(* Logix 5000 project; controller reports 1756-L63 rev 20.11; software revision 20.04; part 25 of 52 *)

        [1708].log_data[0].total := 300.0, [1708].log_data[0].time := 300.0, [1708].log_data[0].minminute := 40, [1708].log_data[0].maxminute := 40, [1708].log_data[0].valid := 1, [1708].log_data[1].valid := 1, [1708].log_data[2].valid := 1, [1708].log_data[3].valid := 1, [1708].log_data[4].valid := 1, [1708].log_data[5].valid := 1, [1708].log_data[6].valid := 1, [1708].log_data[7].valid := 1, [1708].log_data[8].valid := 1, [1708].log_data[9].valid := 1, [1708].log_data[10].valid := 1, [1708].log_data[11].valid := 1, [1708].log_data[12].valid := 1, [1708].log_data[13].valid := 1, [1708].log_data[14].valid := 1, [1708].log_data[15].valid := 1, [1708].log_data[16].valid := 1, [1708].log_data[17].valid := 1, [1708].log_data[18].valid := 1, [1708].log_data[19].valid := 1, [1708].time.Year := 2023, [1708].time.Month := 1, [1708].time.Day := 15, [1708].time.Hour := 14, [1708].time.Minute := 44, [1708].time.Second := 59, [1709].log_data[0].min := 1.0, [1709].log_data[0].max := 1.0, [1709].log_data[0].total := 300.0, [1709].log_data[0].time := 300.0, [1709].log_data[0].minminute := 45, [1709].log_data[0].maxminute := 45, [1709].log_data[0].valid := 1, [1709].log_data[1].valid := 1, [1709].log_data[2].valid := 1, [1709].log_data[3].valid := 1, [1709].log_data[4].valid := 1, [1709].log_data[5].valid := 1, [1709].log_data[6].valid := 1, [1709].log_data[7].valid := 1, [1709].log_data[8].valid := 1, [1709].log_data[9].valid := 1, [1709].log_data[10].valid := 1, [1709].log_data[11].valid := 1, [1709].log_data[12].valid := 1, [1709].log_data[13].valid := 1, [1709].log_data[14].valid := 1, [1709].log_data[15].valid := 1, [1709].log_data[16].valid := 1, [1709].log_data[17].valid := 1, [1709].log_data[18].valid := 1, [1709].log_data[19].valid := 1, [1709].time.Year := 2023, [1709].time.Month := 1, [1709].time.Day := 15, [1709].time.Hour := 14,
        [1709].time.Minute := 49, [1709].time.Second := 59, [1710].log_data[0].min := 1.0, [1710].log_data[0].max := 1.0, [1710].log_data[0].total := 300.0, [1710].log_data[0].time := 300.0, [1710].log_data[0].minminute := 50, [1710].log_data[0].maxminute := 50, [1710].log_data[0].valid := 1, [1710].log_data[1].valid := 1, [1710].log_data[2].valid := 1, [1710].log_data[3].valid := 1, [1710].log_data[4].valid := 1, [1710].log_data[5].valid := 1, [1710].log_data[6].valid := 1, [1710].log_data[7].valid := 1, [1710].log_data[8].valid := 1, [1710].log_data[9].valid := 1, [1710].log_data[10].valid := 1, [1710].log_data[11].valid := 1, [1710].log_data[12].valid := 1, [1710].log_data[13].valid := 1, [1710].log_data[14].valid := 1, [1710].log_data[15].valid := 1, [1710].log_data[16].valid := 1, [1710].log_data[17].valid := 1, [1710].log_data[18].valid := 1, [1710].log_data[19].valid := 1, [1710].time.Year := 2023, [1710].time.Month := 1, [1710].time.Day := 15, [1710].time.Hour := 14, [1710].time.Minute := 54, [1710].time.Second := 59, [1711].log_data[0].min := 1.0, [1711].log_data[0].max := 1.0, [1711].log_data[0].total := 300.0, [1711].log_data[0].time := 300.0, [1711].log_data[0].minminute := 55, [1711].log_data[0].maxminute := 55, [1711].log_data[0].valid := 1, [1711].log_data[1].valid := 1, [1711].log_data[2].valid := 1, [1711].log_data[3].valid := 1, [1711].log_data[4].valid := 1, [1711].log_data[5].valid := 1, [1711].log_data[6].valid := 1, [1711].log_data[7].valid := 1, [1711].log_data[8].valid := 1, [1711].log_data[9].valid := 1, [1711].log_data[10].valid := 1, [1711].log_data[11].valid := 1, [1711].log_data[12].valid := 1, [1711].log_data[13].valid := 1, [1711].log_data[14].valid := 1, [1711].log_data[15].valid := 1, [1711].log_data[16].valid := 1, [1711].log_data[17].valid := 1, [1711].log_data[18].valid := 1, [1711].log_data[19].valid := 1,
        [1711].time.Year := 2023, [1711].time.Month := 1, [1711].time.Day := 15, [1711].time.Hour := 14, [1711].time.Minute := 59, [1711].time.Second := 59, [1712].log_data[0].min := 1.0, [1712].log_data[0].max := 1.0, [1712].log_data[0].total := 300.0, [1712].log_data[0].time := 300.0, [1712].log_data[0].valid := 1, [1712].log_data[1].valid := 1, [1712].log_data[2].valid := 1, [1712].log_data[3].valid := 1, [1712].log_data[4].valid := 1, [1712].log_data[5].valid := 1, [1712].log_data[6].valid := 1, [1712].log_data[7].valid := 1, [1712].log_data[8].valid := 1, [1712].log_data[9].valid := 1, [1712].log_data[10].valid := 1, [1712].log_data[11].valid := 1, [1712].log_data[12].valid := 1, [1712].log_data[13].valid := 1, [1712].log_data[14].valid := 1, [1712].log_data[15].valid := 1, [1712].log_data[16].valid := 1, [1712].log_data[17].valid := 1, [1712].log_data[18].valid := 1, [1712].log_data[19].valid := 1, [1712].time.Year := 2023, [1712].time.Month := 1, [1712].time.Day := 15, [1712].time.Hour := 15, [1712].time.Minute := 4, [1712].time.Second := 59, [1713].log_data[0].min := 1.0, [1713].log_data[0].max := 1.0, [1713].log_data[0].total := 300.0, [1713].log_data[0].time := 300.0, [1713].log_data[0].minminute := 5, [1713].log_data[0].maxminute := 5, [1713].log_data[0].valid := 1, [1713].log_data[1].valid := 1, [1713].log_data[2].valid := 1, [1713].log_data[3].valid := 1, [1713].log_data[4].valid := 1, [1713].log_data[5].valid := 1, [1713].log_data[6].valid := 1, [1713].log_data[7].valid := 1, [1713].log_data[8].valid := 1, [1713].log_data[9].valid := 1, [1713].log_data[10].valid := 1, [1713].log_data[11].valid := 1, [1713].log_data[12].valid := 1, [1713].log_data[13].valid := 1, [1713].log_data[14].valid := 1, [1713].log_data[15].valid := 1, [1713].log_data[16].valid := 1, [1713].log_data[17].valid := 1,
        [1713].log_data[18].valid := 1, [1713].log_data[19].valid := 1, [1713].time.Year := 2023, [1713].time.Month := 1, [1713].time.Day := 15, [1713].time.Hour := 15, [1713].time.Minute := 9, [1713].time.Second := 59, [1714].log_data[0].min := 1.0, [1714].log_data[0].max := 1.0, [1714].log_data[0].total := 300.0, [1714].log_data[0].time := 300.0, [1714].log_data[0].minminute := 10, [1714].log_data[0].maxminute := 10, [1714].log_data[0].valid := 1, [1714].log_data[1].valid := 1, [1714].log_data[2].valid := 1, [1714].log_data[3].valid := 1, [1714].log_data[4].valid := 1, [1714].log_data[5].valid := 1, [1714].log_data[6].valid := 1, [1714].log_data[7].valid := 1, [1714].log_data[8].valid := 1, [1714].log_data[9].valid := 1, [1714].log_data[10].valid := 1, [1714].log_data[11].valid := 1, [1714].log_data[12].valid := 1, [1714].log_data[13].valid := 1, [1714].log_data[14].valid := 1, [1714].log_data[15].valid := 1, [1714].log_data[16].valid := 1, [1714].log_data[17].valid := 1, [1714].log_data[18].valid := 1, [1714].log_data[19].valid := 1, [1714].time.Year := 2023, [1714].time.Month := 1, [1714].time.Day := 15, [1714].time.Hour := 15, [1714].time.Minute := 14, [1714].time.Second := 59, [1715].log_data[0].min := 1.0, [1715].log_data[0].max := 1.0, [1715].log_data[0].total := 300.0, [1715].log_data[0].time := 300.0, [1715].log_data[0].minminute := 15, [1715].log_data[0].maxminute := 15, [1715].log_data[0].valid := 1, [1715].log_data[1].valid := 1, [1715].log_data[2].valid := 1, [1715].log_data[3].valid := 1, [1715].log_data[4].valid := 1, [1715].log_data[5].valid := 1, [1715].log_data[6].valid := 1, [1715].log_data[7].valid := 1, [1715].log_data[8].valid := 1, [1715].log_data[9].valid := 1, [1715].log_data[10].valid := 1, [1715].log_data[11].valid := 1, [1715].log_data[12].valid := 1, [1715].log_data[13].valid := 1,
        [1715].log_data[14].valid := 1, [1715].log_data[15].valid := 1, [1715].log_data[16].valid := 1, [1715].log_data[17].valid := 1, [1715].log_data[18].valid := 1, [1715].log_data[19].valid := 1, [1715].time.Year := 2023, [1715].time.Month := 1, [1715].time.Day := 15, [1715].time.Hour := 15, [1715].time.Minute := 19, [1715].time.Second := 59, [1716].log_data[0].min := 1.0, [1716].log_data[0].max := 1.0, [1716].log_data[0].total := 300.0, [1716].log_data[0].time := 300.0, [1716].log_data[0].minminute := 20, [1716].log_data[0].maxminute := 20, [1716].log_data[0].valid := 1, [1716].log_data[1].valid := 1, [1716].log_data[2].valid := 1, [1716].log_data[3].valid := 1, [1716].log_data[4].valid := 1, [1716].log_data[5].valid := 1, [1716].log_data[6].valid := 1, [1716].log_data[7].valid := 1, [1716].log_data[8].valid := 1, [1716].log_data[9].valid := 1, [1716].log_data[10].valid := 1, [1716].log_data[11].valid := 1, [1716].log_data[12].valid := 1, [1716].log_data[13].valid := 1, [1716].log_data[14].valid := 1, [1716].log_data[15].valid := 1, [1716].log_data[16].valid := 1, [1716].log_data[17].valid := 1, [1716].log_data[18].valid := 1, [1716].log_data[19].valid := 1, [1716].time.Year := 2023, [1716].time.Month := 1, [1716].time.Day := 15, [1716].time.Hour := 15, [1716].time.Minute := 24, [1716].time.Second := 59, [1717].log_data[0].min := 1.0, [1717].log_data[0].max := 1.0, [1717].log_data[0].total := 300.0, [1717].log_data[0].time := 300.0, [1717].log_data[0].minminute := 25, [1717].log_data[0].maxminute := 25, [1717].log_data[0].valid := 1, [1717].log_data[1].valid := 1, [1717].log_data[2].valid := 1, [1717].log_data[3].valid := 1, [1717].log_data[4].valid := 1, [1717].log_data[5].valid := 1, [1717].log_data[6].valid := 1, [1717].log_data[7].valid := 1, [1717].log_data[8].valid := 1, [1717].log_data[9].valid := 1,
        [1717].log_data[10].valid := 1, [1717].log_data[11].valid := 1, [1717].log_data[12].valid := 1, [1717].log_data[13].valid := 1, [1717].log_data[14].valid := 1, [1717].log_data[15].valid := 1, [1717].log_data[16].valid := 1, [1717].log_data[17].valid := 1, [1717].log_data[18].valid := 1, [1717].log_data[19].valid := 1, [1717].time.Year := 2023, [1717].time.Month := 1, [1717].time.Day := 15, [1717].time.Hour := 15, [1717].time.Minute := 29, [1717].time.Second := 59, [1718].log_data[0].min := 1.0, [1718].log_data[0].max := 1.0, [1718].log_data[0].total := 300.0, [1718].log_data[0].time := 300.0, [1718].log_data[0].minminute := 30, [1718].log_data[0].maxminute := 30, [1718].log_data[0].valid := 1, [1718].log_data[1].valid := 1, [1718].log_data[2].valid := 1, [1718].log_data[3].valid := 1, [1718].log_data[4].valid := 1, [1718].log_data[5].valid := 1, [1718].log_data[6].valid := 1, [1718].log_data[7].valid := 1, [1718].log_data[8].valid := 1, [1718].log_data[9].valid := 1, [1718].log_data[10].valid := 1, [1718].log_data[11].valid := 1, [1718].log_data[12].valid := 1, [1718].log_data[13].valid := 1, [1718].log_data[14].valid := 1, [1718].log_data[15].valid := 1, [1718].log_data[16].valid := 1, [1718].log_data[17].valid := 1, [1718].log_data[18].valid := 1, [1718].log_data[19].valid := 1, [1718].time.Year := 2023, [1718].time.Month := 1, [1718].time.Day := 15, [1718].time.Hour := 15, [1718].time.Minute := 34, [1718].time.Second := 59, [1719].log_data[0].min := 1.0, [1719].log_data[0].max := 1.0, [1719].log_data[0].total := 300.0, [1719].log_data[0].time := 300.0, [1719].log_data[0].minminute := 35, [1719].log_data[0].maxminute := 35, [1719].log_data[0].valid := 1, [1719].log_data[1].valid := 1, [1719].log_data[2].valid := 1, [1719].log_data[3].valid := 1, [1719].log_data[4].valid := 1, [1719].log_data[5].valid := 1,
        [1719].log_data[6].valid := 1, [1719].log_data[7].valid := 1, [1719].log_data[8].valid := 1, [1719].log_data[9].valid := 1, [1719].log_data[10].valid := 1, [1719].log_data[11].valid := 1, [1719].log_data[12].valid := 1, [1719].log_data[13].valid := 1, [1719].log_data[14].valid := 1, [1719].log_data[15].valid := 1, [1719].log_data[16].valid := 1, [1719].log_data[17].valid := 1, [1719].log_data[18].valid := 1, [1719].log_data[19].valid := 1, [1719].time.Year := 2023, [1719].time.Month := 1, [1719].time.Day := 15, [1719].time.Hour := 15, [1719].time.Minute := 39, [1719].time.Second := 59, [1720].log_data[0].min := 1.0, [1720].log_data[0].max := 1.0, [1720].log_data[0].total := 300.0, [1720].log_data[0].time := 300.0, [1720].log_data[0].minminute := 40, [1720].log_data[0].maxminute := 40, [1720].log_data[0].valid := 1, [1720].log_data[1].valid := 1, [1720].log_data[2].valid := 1, [1720].log_data[3].valid := 1, [1720].log_data[4].valid := 1, [1720].log_data[5].valid := 1, [1720].log_data[6].valid := 1, [1720].log_data[7].valid := 1, [1720].log_data[8].valid := 1, [1720].log_data[9].valid := 1, [1720].log_data[10].valid := 1, [1720].log_data[11].valid := 1, [1720].log_data[12].valid := 1, [1720].log_data[13].valid := 1, [1720].log_data[14].valid := 1, [1720].log_data[15].valid := 1, [1720].log_data[16].valid := 1, [1720].log_data[17].valid := 1, [1720].log_data[18].valid := 1, [1720].log_data[19].valid := 1, [1720].time.Year := 2023, [1720].time.Month := 1, [1720].time.Day := 15, [1720].time.Hour := 15, [1720].time.Minute := 44, [1720].time.Second := 59, [1721].log_data[0].min := 1.0, [1721].log_data[0].max := 1.0, [1721].log_data[0].total := 300.0, [1721].log_data[0].time := 300.0, [1721].log_data[0].minminute := 45, [1721].log_data[0].maxminute := 45, [1721].log_data[0].valid := 1, [1721].log_data[1].valid := 1,
        [1721].log_data[2].valid := 1, [1721].log_data[3].valid := 1, [1721].log_data[4].valid := 1, [1721].log_data[5].valid := 1, [1721].log_data[6].valid := 1, [1721].log_data[7].valid := 1, [1721].log_data[8].valid := 1, [1721].log_data[9].valid := 1, [1721].log_data[10].valid := 1, [1721].log_data[11].valid := 1, [1721].log_data[12].valid := 1, [1721].log_data[13].valid := 1, [1721].log_data[14].valid := 1, [1721].log_data[15].valid := 1, [1721].log_data[16].valid := 1, [1721].log_data[17].valid := 1, [1721].log_data[18].valid := 1, [1721].log_data[19].valid := 1, [1721].time.Year := 2023, [1721].time.Month := 1, [1721].time.Day := 15, [1721].time.Hour := 15, [1721].time.Minute := 49, [1721].time.Second := 59, [1722].log_data[0].min := 1.0, [1722].log_data[0].max := 1.0, [1722].log_data[0].total := 300.0, [1722].log_data[0].time := 300.0, [1722].log_data[0].minminute := 50, [1722].log_data[0].maxminute := 50, [1722].log_data[0].valid := 1, [1722].log_data[1].valid := 1, [1722].log_data[2].valid := 1, [1722].log_data[3].valid := 1, [1722].log_data[4].valid := 1, [1722].log_data[5].valid := 1, [1722].log_data[6].valid := 1, [1722].log_data[7].valid := 1, [1722].log_data[8].valid := 1, [1722].log_data[9].valid := 1, [1722].log_data[10].valid := 1, [1722].log_data[11].valid := 1, [1722].log_data[12].valid := 1, [1722].log_data[13].valid := 1, [1722].log_data[14].valid := 1, [1722].log_data[15].valid := 1, [1722].log_data[16].valid := 1, [1722].log_data[17].valid := 1, [1722].log_data[18].valid := 1, [1722].log_data[19].valid := 1, [1722].time.Year := 2023, [1722].time.Month := 1, [1722].time.Day := 15, [1722].time.Hour := 15, [1722].time.Minute := 54, [1722].time.Second := 59, [1723].log_data[0].min := 1.0, [1723].log_data[0].max := 1.0, [1723].log_data[0].total := 300.0, [1723].log_data[0].time := 300.0,
        [1723].log_data[0].minminute := 55, [1723].log_data[0].maxminute := 55, [1723].log_data[0].valid := 1, [1723].log_data[1].valid := 1, [1723].log_data[2].valid := 1, [1723].log_data[3].valid := 1, [1723].log_data[4].valid := 1, [1723].log_data[5].valid := 1, [1723].log_data[6].valid := 1, [1723].log_data[7].valid := 1, [1723].log_data[8].valid := 1, [1723].log_data[9].valid := 1, [1723].log_data[10].valid := 1, [1723].log_data[11].valid := 1, [1723].log_data[12].valid := 1, [1723].log_data[13].valid := 1, [1723].log_data[14].valid := 1, [1723].log_data[15].valid := 1, [1723].log_data[16].valid := 1, [1723].log_data[17].valid := 1, [1723].log_data[18].valid := 1, [1723].log_data[19].valid := 1, [1723].time.Year := 2023, [1723].time.Month := 1, [1723].time.Day := 15, [1723].time.Hour := 15, [1723].time.Minute := 59, [1723].time.Second := 59, [1724].log_data[0].min := 1.0, [1724].log_data[0].max := 1.0, [1724].log_data[0].total := 300.0, [1724].log_data[0].time := 300.0, [1724].log_data[0].valid := 1, [1724].log_data[1].valid := 1, [1724].log_data[2].valid := 1, [1724].log_data[3].valid := 1, [1724].log_data[4].valid := 1, [1724].log_data[5].valid := 1, [1724].log_data[6].valid := 1, [1724].log_data[7].valid := 1, [1724].log_data[8].valid := 1, [1724].log_data[9].valid := 1, [1724].log_data[10].valid := 1, [1724].log_data[11].valid := 1, [1724].log_data[12].valid := 1, [1724].log_data[13].valid := 1, [1724].log_data[14].valid := 1, [1724].log_data[15].valid := 1, [1724].log_data[16].valid := 1, [1724].log_data[17].valid := 1, [1724].log_data[18].valid := 1, [1724].log_data[19].valid := 1, [1724].time.Year := 2023, [1724].time.Month := 1, [1724].time.Day := 15, [1724].time.Hour := 16, [1724].time.Minute := 4, [1724].time.Second := 59, [1725].log_data[0].min := 1.0, [1725].log_data[0].max := 1.0,
        [1725].log_data[0].total := 300.0, [1725].log_data[0].time := 300.0, [1725].log_data[0].minminute := 5, [1725].log_data[0].maxminute := 5, [1725].log_data[0].valid := 1, [1725].log_data[1].valid := 1, [1725].log_data[2].valid := 1, [1725].log_data[3].valid := 1, [1725].log_data[4].valid := 1, [1725].log_data[5].valid := 1, [1725].log_data[6].valid := 1, [1725].log_data[7].valid := 1, [1725].log_data[8].valid := 1, [1725].log_data[9].valid := 1, [1725].log_data[10].valid := 1, [1725].log_data[11].valid := 1, [1725].log_data[12].valid := 1, [1725].log_data[13].valid := 1, [1725].log_data[14].valid := 1, [1725].log_data[15].valid := 1, [1725].log_data[16].valid := 1, [1725].log_data[17].valid := 1, [1725].log_data[18].valid := 1, [1725].log_data[19].valid := 1, [1725].time.Year := 2023, [1725].time.Month := 1, [1725].time.Day := 15, [1725].time.Hour := 16, [1725].time.Minute := 9, [1725].time.Second := 59, [1726].log_data[0].min := 1.0, [1726].log_data[0].max := 1.0, [1726].log_data[0].total := 300.0, [1726].log_data[0].time := 300.0, [1726].log_data[0].minminute := 10, [1726].log_data[0].maxminute := 10, [1726].log_data[0].valid := 1, [1726].log_data[1].valid := 1, [1726].log_data[2].valid := 1, [1726].log_data[3].valid := 1, [1726].log_data[4].valid := 1, [1726].log_data[5].valid := 1, [1726].log_data[6].valid := 1, [1726].log_data[7].valid := 1, [1726].log_data[8].valid := 1, [1726].log_data[9].valid := 1, [1726].log_data[10].valid := 1, [1726].log_data[11].valid := 1, [1726].log_data[12].valid := 1, [1726].log_data[13].valid := 1, [1726].log_data[14].valid := 1, [1726].log_data[15].valid := 1, [1726].log_data[16].valid := 1, [1726].log_data[17].valid := 1, [1726].log_data[18].valid := 1, [1726].log_data[19].valid := 1, [1726].time.Year := 2023, [1726].time.Month := 1, [1726].time.Day := 15, [1726].time.Hour := 16,
        [1726].time.Minute := 14, [1726].time.Second := 59, [1727].log_data[0].min := 1.0, [1727].log_data[0].max := 1.0, [1727].log_data[0].total := 300.0, [1727].log_data[0].time := 300.0, [1727].log_data[0].minminute := 15, [1727].log_data[0].maxminute := 15, [1727].log_data[0].valid := 1, [1727].log_data[1].valid := 1, [1727].log_data[2].valid := 1, [1727].log_data[3].valid := 1, [1727].log_data[4].valid := 1, [1727].log_data[5].valid := 1, [1727].log_data[6].valid := 1, [1727].log_data[7].valid := 1, [1727].log_data[8].valid := 1, [1727].log_data[9].valid := 1, [1727].log_data[10].valid := 1, [1727].log_data[11].valid := 1, [1727].log_data[12].valid := 1, [1727].log_data[13].valid := 1, [1727].log_data[14].valid := 1, [1727].log_data[15].valid := 1, [1727].log_data[16].valid := 1, [1727].log_data[17].valid := 1, [1727].log_data[18].valid := 1, [1727].log_data[19].valid := 1, [1727].time.Year := 2023, [1727].time.Month := 1, [1727].time.Day := 15, [1727].time.Hour := 16, [1727].time.Minute := 19, [1727].time.Second := 59, [1728].log_data[0].min := 1.0, [1728].log_data[0].max := 1.0, [1728].log_data[0].total := 300.0, [1728].log_data[0].time := 300.0, [1728].log_data[0].minminute := 20, [1728].log_data[0].maxminute := 20, [1728].log_data[0].valid := 1, [1728].log_data[1].valid := 1, [1728].log_data[2].valid := 1, [1728].log_data[3].valid := 1, [1728].log_data[4].valid := 1, [1728].log_data[5].valid := 1, [1728].log_data[6].valid := 1, [1728].log_data[7].valid := 1, [1728].log_data[8].valid := 1, [1728].log_data[9].valid := 1, [1728].log_data[10].valid := 1, [1728].log_data[11].valid := 1, [1728].log_data[12].valid := 1, [1728].log_data[13].valid := 1, [1728].log_data[14].valid := 1, [1728].log_data[15].valid := 1, [1728].log_data[16].valid := 1, [1728].log_data[17].valid := 1, [1728].log_data[18].valid := 1, [1728].log_data[19].valid := 1,
        [1728].time.Year := 2023, [1728].time.Month := 1, [1728].time.Day := 15, [1728].time.Hour := 16, [1728].time.Minute := 24, [1728].time.Second := 59, [1729].log_data[0].min := 1.0, [1729].log_data[0].max := 1.0, [1729].log_data[0].total := 300.0, [1729].log_data[0].time := 300.0, [1729].log_data[0].minminute := 25, [1729].log_data[0].maxminute := 25, [1729].log_data[0].valid := 1, [1729].log_data[1].valid := 1, [1729].log_data[2].valid := 1, [1729].log_data[3].valid := 1, [1729].log_data[4].valid := 1, [1729].log_data[5].valid := 1, [1729].log_data[6].valid := 1, [1729].log_data[7].valid := 1, [1729].log_data[8].valid := 1, [1729].log_data[9].valid := 1, [1729].log_data[10].valid := 1, [1729].log_data[11].valid := 1, [1729].log_data[12].valid := 1, [1729].log_data[13].valid := 1, [1729].log_data[14].valid := 1, [1729].log_data[15].valid := 1, [1729].log_data[16].valid := 1, [1729].log_data[17].valid := 1, [1729].log_data[18].valid := 1, [1729].log_data[19].valid := 1, [1729].time.Year := 2023, [1729].time.Month := 1, [1729].time.Day := 15, [1729].time.Hour := 16, [1729].time.Minute := 29, [1729].time.Second := 59, [1730].log_data[0].min := 1.0, [1730].log_data[0].max := 1.0, [1730].log_data[0].total := 300.0, [1730].log_data[0].time := 300.0, [1730].log_data[0].minminute := 30, [1730].log_data[0].maxminute := 30, [1730].log_data[0].valid := 1, [1730].log_data[1].valid := 1, [1730].log_data[2].valid := 1, [1730].log_data[3].valid := 1, [1730].log_data[4].valid := 1, [1730].log_data[5].valid := 1, [1730].log_data[6].valid := 1, [1730].log_data[7].valid := 1, [1730].log_data[8].valid := 1, [1730].log_data[9].valid := 1, [1730].log_data[10].valid := 1, [1730].log_data[11].valid := 1, [1730].log_data[12].valid := 1, [1730].log_data[13].valid := 1, [1730].log_data[14].valid := 1, [1730].log_data[15].valid := 1,
        [1730].log_data[16].valid := 1, [1730].log_data[17].valid := 1, [1730].log_data[18].valid := 1, [1730].log_data[19].valid := 1, [1730].time.Year := 2023, [1730].time.Month := 1, [1730].time.Day := 15, [1730].time.Hour := 16, [1730].time.Minute := 34, [1730].time.Second := 59, [1731].log_data[0].min := 1.0, [1731].log_data[0].max := 1.0, [1731].log_data[0].total := 300.0, [1731].log_data[0].time := 300.0, [1731].log_data[0].minminute := 35, [1731].log_data[0].maxminute := 35, [1731].log_data[0].valid := 1, [1731].log_data[1].valid := 1, [1731].log_data[2].valid := 1, [1731].log_data[3].valid := 1, [1731].log_data[4].valid := 1, [1731].log_data[5].valid := 1, [1731].log_data[6].valid := 1, [1731].log_data[7].valid := 1, [1731].log_data[8].valid := 1, [1731].log_data[9].valid := 1, [1731].log_data[10].valid := 1, [1731].log_data[11].valid := 1, [1731].log_data[12].valid := 1, [1731].log_data[13].valid := 1, [1731].log_data[14].valid := 1, [1731].log_data[15].valid := 1, [1731].log_data[16].valid := 1, [1731].log_data[17].valid := 1, [1731].log_data[18].valid := 1, [1731].log_data[19].valid := 1, [1731].time.Year := 2023, [1731].time.Month := 1, [1731].time.Day := 15, [1731].time.Hour := 16, [1731].time.Minute := 39, [1731].time.Second := 59, [1732].log_data[0].min := 1.0, [1732].log_data[0].max := 1.0, [1732].log_data[0].total := 300.0, [1732].log_data[0].time := 300.0, [1732].log_data[0].minminute := 40, [1732].log_data[0].maxminute := 40, [1732].log_data[0].valid := 1, [1732].log_data[1].valid := 1, [1732].log_data[2].valid := 1, [1732].log_data[3].valid := 1, [1732].log_data[4].valid := 1, [1732].log_data[5].valid := 1, [1732].log_data[6].valid := 1, [1732].log_data[7].valid := 1, [1732].log_data[8].valid := 1, [1732].log_data[9].valid := 1, [1732].log_data[10].valid := 1, [1732].log_data[11].valid := 1,
        [1732].log_data[12].valid := 1, [1732].log_data[13].valid := 1, [1732].log_data[14].valid := 1, [1732].log_data[15].valid := 1, [1732].log_data[16].valid := 1, [1732].log_data[17].valid := 1, [1732].log_data[18].valid := 1, [1732].log_data[19].valid := 1, [1732].time.Year := 2023, [1732].time.Month := 1, [1732].time.Day := 15, [1732].time.Hour := 16, [1732].time.Minute := 44, [1732].time.Second := 59, [1733].log_data[0].min := 1.0, [1733].log_data[0].max := 1.0, [1733].log_data[0].total := 300.0, [1733].log_data[0].time := 300.0, [1733].log_data[0].minminute := 45, [1733].log_data[0].maxminute := 45, [1733].log_data[0].valid := 1, [1733].log_data[1].valid := 1, [1733].log_data[2].valid := 1, [1733].log_data[3].valid := 1, [1733].log_data[4].valid := 1, [1733].log_data[5].valid := 1, [1733].log_data[6].valid := 1, [1733].log_data[7].valid := 1, [1733].log_data[8].valid := 1, [1733].log_data[9].valid := 1, [1733].log_data[10].valid := 1, [1733].log_data[11].valid := 1, [1733].log_data[12].valid := 1, [1733].log_data[13].valid := 1, [1733].log_data[14].valid := 1, [1733].log_data[15].valid := 1, [1733].log_data[16].valid := 1, [1733].log_data[17].valid := 1, [1733].log_data[18].valid := 1, [1733].log_data[19].valid := 1, [1733].time.Year := 2023, [1733].time.Month := 1, [1733].time.Day := 15, [1733].time.Hour := 16, [1733].time.Minute := 49, [1733].time.Second := 59, [1734].log_data[0].min := 1.0, [1734].log_data[0].max := 1.0, [1734].log_data[0].total := 300.0, [1734].log_data[0].time := 300.0, [1734].log_data[0].minminute := 50, [1734].log_data[0].maxminute := 50, [1734].log_data[0].valid := 1, [1734].log_data[1].valid := 1, [1734].log_data[2].valid := 1, [1734].log_data[3].valid := 1, [1734].log_data[4].valid := 1, [1734].log_data[5].valid := 1, [1734].log_data[6].valid := 1, [1734].log_data[7].valid := 1,
        [1734].log_data[8].valid := 1, [1734].log_data[9].valid := 1, [1734].log_data[10].valid := 1, [1734].log_data[11].valid := 1, [1734].log_data[12].valid := 1, [1734].log_data[13].valid := 1, [1734].log_data[14].valid := 1, [1734].log_data[15].valid := 1, [1734].log_data[16].valid := 1, [1734].log_data[17].valid := 1, [1734].log_data[18].valid := 1, [1734].log_data[19].valid := 1, [1734].time.Year := 2023, [1734].time.Month := 1, [1734].time.Day := 15, [1734].time.Hour := 16, [1734].time.Minute := 54, [1734].time.Second := 59, [1735].log_data[0].min := 1.0, [1735].log_data[0].max := 1.0, [1735].log_data[0].total := 300.0, [1735].log_data[0].time := 300.0, [1735].log_data[0].minminute := 55, [1735].log_data[0].maxminute := 55, [1735].log_data[0].valid := 1, [1735].log_data[1].valid := 1, [1735].log_data[2].valid := 1, [1735].log_data[3].valid := 1, [1735].log_data[4].valid := 1, [1735].log_data[5].valid := 1, [1735].log_data[6].valid := 1, [1735].log_data[7].valid := 1, [1735].log_data[8].valid := 1, [1735].log_data[9].valid := 1, [1735].log_data[10].valid := 1, [1735].log_data[11].valid := 1, [1735].log_data[12].valid := 1, [1735].log_data[13].valid := 1, [1735].log_data[14].valid := 1, [1735].log_data[15].valid := 1, [1735].log_data[16].valid := 1, [1735].log_data[17].valid := 1, [1735].log_data[18].valid := 1, [1735].log_data[19].valid := 1, [1735].time.Year := 2023, [1735].time.Month := 1, [1735].time.Day := 15, [1735].time.Hour := 16, [1735].time.Minute := 59, [1735].time.Second := 59, [1736].log_data[0].min := 1.0, [1736].log_data[0].max := 1.0, [1736].log_data[0].total := 300.0, [1736].log_data[0].time := 300.0, [1736].log_data[0].valid := 1, [1736].log_data[1].valid := 1, [1736].log_data[2].valid := 1, [1736].log_data[3].valid := 1, [1736].log_data[4].valid := 1, [1736].log_data[5].valid := 1,
        [1736].log_data[6].valid := 1, [1736].log_data[7].valid := 1, [1736].log_data[8].valid := 1, [1736].log_data[9].valid := 1, [1736].log_data[10].valid := 1, [1736].log_data[11].valid := 1, [1736].log_data[12].valid := 1, [1736].log_data[13].valid := 1, [1736].log_data[14].valid := 1, [1736].log_data[15].valid := 1, [1736].log_data[16].valid := 1, [1736].log_data[17].valid := 1, [1736].log_data[18].valid := 1, [1736].log_data[19].valid := 1, [1736].time.Year := 2023, [1736].time.Month := 1, [1736].time.Day := 15, [1736].time.Hour := 17, [1736].time.Minute := 4, [1736].time.Second := 59, [1737].log_data[0].min := 1.0, [1737].log_data[0].max := 1.0, [1737].log_data[0].total := 300.0, [1737].log_data[0].time := 300.0, [1737].log_data[0].minminute := 5, [1737].log_data[0].maxminute := 5, [1737].log_data[0].valid := 1, [1737].log_data[1].valid := 1, [1737].log_data[2].valid := 1, [1737].log_data[3].valid := 1, [1737].log_data[4].valid := 1, [1737].log_data[5].valid := 1, [1737].log_data[6].valid := 1, [1737].log_data[7].valid := 1, [1737].log_data[8].valid := 1, [1737].log_data[9].valid := 1, [1737].log_data[10].valid := 1, [1737].log_data[11].valid := 1, [1737].log_data[12].valid := 1, [1737].log_data[13].valid := 1, [1737].log_data[14].valid := 1, [1737].log_data[15].valid := 1, [1737].log_data[16].valid := 1, [1737].log_data[17].valid := 1, [1737].log_data[18].valid := 1, [1737].log_data[19].valid := 1, [1737].time.Year := 2023, [1737].time.Month := 1, [1737].time.Day := 15, [1737].time.Hour := 17, [1737].time.Minute := 9, [1737].time.Second := 59, [1738].log_data[0].min := 1.0, [1738].log_data[0].max := 1.0, [1738].log_data[0].total := 300.0, [1738].log_data[0].time := 300.0, [1738].log_data[0].minminute := 10, [1738].log_data[0].maxminute := 10, [1738].log_data[0].valid := 1, [1738].log_data[1].valid := 1,
        [1738].log_data[2].valid := 1, [1738].log_data[3].valid := 1, [1738].log_data[4].valid := 1, [1738].log_data[5].valid := 1, [1738].log_data[6].valid := 1, [1738].log_data[7].valid := 1, [1738].log_data[8].valid := 1, [1738].log_data[9].valid := 1, [1738].log_data[10].valid := 1, [1738].log_data[11].valid := 1, [1738].log_data[12].valid := 1, [1738].log_data[13].valid := 1, [1738].log_data[14].valid := 1, [1738].log_data[15].valid := 1, [1738].log_data[16].valid := 1, [1738].log_data[17].valid := 1, [1738].log_data[18].valid := 1, [1738].log_data[19].valid := 1, [1738].time.Year := 2023, [1738].time.Month := 1, [1738].time.Day := 15, [1738].time.Hour := 17, [1738].time.Minute := 14, [1738].time.Second := 59, [1739].log_data[0].min := 1.0, [1739].log_data[0].max := 1.0, [1739].log_data[0].total := 300.0, [1739].log_data[0].time := 300.0, [1739].log_data[0].minminute := 15, [1739].log_data[0].maxminute := 15, [1739].log_data[0].valid := 1, [1739].log_data[1].valid := 1, [1739].log_data[2].valid := 1, [1739].log_data[3].valid := 1, [1739].log_data[4].valid := 1, [1739].log_data[5].valid := 1, [1739].log_data[6].valid := 1, [1739].log_data[7].valid := 1, [1739].log_data[8].valid := 1, [1739].log_data[9].valid := 1, [1739].log_data[10].valid := 1, [1739].log_data[11].valid := 1, [1739].log_data[12].valid := 1, [1739].log_data[13].valid := 1, [1739].log_data[14].valid := 1, [1739].log_data[15].valid := 1, [1739].log_data[16].valid := 1, [1739].log_data[17].valid := 1, [1739].log_data[18].valid := 1, [1739].log_data[19].valid := 1, [1739].time.Year := 2023, [1739].time.Month := 1, [1739].time.Day := 15, [1739].time.Hour := 17, [1739].time.Minute := 19, [1739].time.Second := 59, [1740].log_data[0].min := 1.0, [1740].log_data[0].max := 1.0, [1740].log_data[0].total := 300.0, [1740].log_data[0].time := 300.0,
        [1740].log_data[0].minminute := 20, [1740].log_data[0].maxminute := 20, [1740].log_data[0].valid := 1, [1740].log_data[1].valid := 1, [1740].log_data[2].valid := 1, [1740].log_data[3].valid := 1, [1740].log_data[4].valid := 1, [1740].log_data[5].valid := 1, [1740].log_data[6].valid := 1, [1740].log_data[7].valid := 1, [1740].log_data[8].valid := 1, [1740].log_data[9].valid := 1, [1740].log_data[10].valid := 1, [1740].log_data[11].valid := 1, [1740].log_data[12].valid := 1, [1740].log_data[13].valid := 1, [1740].log_data[14].valid := 1, [1740].log_data[15].valid := 1, [1740].log_data[16].valid := 1, [1740].log_data[17].valid := 1, [1740].log_data[18].valid := 1, [1740].log_data[19].valid := 1, [1740].time.Year := 2023, [1740].time.Month := 1, [1740].time.Day := 15, [1740].time.Hour := 17, [1740].time.Minute := 24, [1740].time.Second := 59, [1741].log_data[0].min := 1.0, [1741].log_data[0].max := 1.0, [1741].log_data[0].total := 300.0, [1741].log_data[0].time := 300.0, [1741].log_data[0].minminute := 25, [1741].log_data[0].maxminute := 25, [1741].log_data[0].valid := 1, [1741].log_data[1].valid := 1, [1741].log_data[2].valid := 1, [1741].log_data[3].valid := 1, [1741].log_data[4].valid := 1, [1741].log_data[5].valid := 1, [1741].log_data[6].valid := 1, [1741].log_data[7].valid := 1, [1741].log_data[8].valid := 1, [1741].log_data[9].valid := 1, [1741].log_data[10].valid := 1, [1741].log_data[11].valid := 1, [1741].log_data[12].valid := 1, [1741].log_data[13].valid := 1, [1741].log_data[14].valid := 1, [1741].log_data[15].valid := 1, [1741].log_data[16].valid := 1, [1741].log_data[17].valid := 1, [1741].log_data[18].valid := 1, [1741].log_data[19].valid := 1, [1741].time.Year := 2023, [1741].time.Month := 1, [1741].time.Day := 15, [1741].time.Hour := 17, [1741].time.Minute := 29, [1741].time.Second := 59,
        [1742].log_data[0].min := 1.0, [1742].log_data[0].max := 1.0, [1742].log_data[0].total := 300.0, [1742].log_data[0].time := 300.0, [1742].log_data[0].minminute := 30, [1742].log_data[0].maxminute := 30, [1742].log_data[0].valid := 1, [1742].log_data[1].valid := 1, [1742].log_data[2].valid := 1, [1742].log_data[3].valid := 1, [1742].log_data[4].valid := 1, [1742].log_data[5].valid := 1, [1742].log_data[6].valid := 1, [1742].log_data[7].valid := 1, [1742].log_data[8].valid := 1, [1742].log_data[9].valid := 1, [1742].log_data[10].valid := 1, [1742].log_data[11].valid := 1, [1742].log_data[12].valid := 1, [1742].log_data[13].valid := 1, [1742].log_data[14].valid := 1, [1742].log_data[15].valid := 1, [1742].log_data[16].valid := 1, [1742].log_data[17].valid := 1, [1742].log_data[18].valid := 1, [1742].log_data[19].valid := 1, [1742].time.Year := 2023, [1742].time.Month := 1, [1742].time.Day := 15, [1742].time.Hour := 17, [1742].time.Minute := 34, [1742].time.Second := 59, [1743].log_data[0].min := 1.0, [1743].log_data[0].max := 1.0, [1743].log_data[0].total := 300.0, [1743].log_data[0].time := 300.0, [1743].log_data[0].minminute := 35, [1743].log_data[0].maxminute := 35, [1743].log_data[0].valid := 1, [1743].log_data[1].valid := 1, [1743].log_data[2].valid := 1, [1743].log_data[3].valid := 1, [1743].log_data[4].valid := 1, [1743].log_data[5].valid := 1, [1743].log_data[6].valid := 1, [1743].log_data[7].valid := 1, [1743].log_data[8].valid := 1, [1743].log_data[9].valid := 1, [1743].log_data[10].valid := 1, [1743].log_data[11].valid := 1, [1743].log_data[12].valid := 1, [1743].log_data[13].valid := 1, [1743].log_data[14].valid := 1, [1743].log_data[15].valid := 1, [1743].log_data[16].valid := 1, [1743].log_data[17].valid := 1, [1743].log_data[18].valid := 1, [1743].log_data[19].valid := 1, [1743].time.Year := 2023, [1743].time.Month := 1,
        [1743].time.Day := 15, [1743].time.Hour := 17, [1743].time.Minute := 39, [1743].time.Second := 59, [1744].log_data[0].min := 1.0, [1744].log_data[0].max := 1.0, [1744].log_data[0].total := 300.0, [1744].log_data[0].time := 300.0, [1744].log_data[0].minminute := 40, [1744].log_data[0].maxminute := 40, [1744].log_data[0].valid := 1, [1744].log_data[1].valid := 1, [1744].log_data[2].valid := 1, [1744].log_data[3].valid := 1, [1744].log_data[4].valid := 1, [1744].log_data[5].valid := 1, [1744].log_data[6].valid := 1, [1744].log_data[7].valid := 1, [1744].log_data[8].valid := 1, [1744].log_data[9].valid := 1, [1744].log_data[10].valid := 1, [1744].log_data[11].valid := 1, [1744].log_data[12].valid := 1, [1744].log_data[13].valid := 1, [1744].log_data[14].valid := 1, [1744].log_data[15].valid := 1, [1744].log_data[16].valid := 1, [1744].log_data[17].valid := 1, [1744].log_data[18].valid := 1, [1744].log_data[19].valid := 1, [1744].time.Year := 2023, [1744].time.Month := 1, [1744].time.Day := 15, [1744].time.Hour := 17, [1744].time.Minute := 44, [1744].time.Second := 59, [1745].log_data[0].min := 1.0, [1745].log_data[0].max := 1.0, [1745].log_data[0].total := 300.0, [1745].log_data[0].time := 300.0, [1745].log_data[0].minminute := 45, [1745].log_data[0].maxminute := 45, [1745].log_data[0].valid := 1, [1745].log_data[1].valid := 1, [1745].log_data[2].valid := 1, [1745].log_data[3].valid := 1, [1745].log_data[4].valid := 1, [1745].log_data[5].valid := 1, [1745].log_data[6].valid := 1, [1745].log_data[7].valid := 1, [1745].log_data[8].valid := 1, [1745].log_data[9].valid := 1, [1745].log_data[10].valid := 1, [1745].log_data[11].valid := 1, [1745].log_data[12].valid := 1, [1745].log_data[13].valid := 1, [1745].log_data[14].valid := 1, [1745].log_data[15].valid := 1, [1745].log_data[16].valid := 1, [1745].log_data[17].valid := 1,
        [1745].log_data[18].valid := 1, [1745].log_data[19].valid := 1, [1745].time.Year := 2023, [1745].time.Month := 1, [1745].time.Day := 15, [1745].time.Hour := 17, [1745].time.Minute := 49, [1745].time.Second := 59, [1746].log_data[0].min := 1.0, [1746].log_data[0].max := 1.0, [1746].log_data[0].total := 300.0, [1746].log_data[0].time := 300.0, [1746].log_data[0].minminute := 50, [1746].log_data[0].maxminute := 50, [1746].log_data[0].valid := 1, [1746].log_data[1].valid := 1, [1746].log_data[2].valid := 1, [1746].log_data[3].valid := 1, [1746].log_data[4].valid := 1, [1746].log_data[5].valid := 1, [1746].log_data[6].valid := 1, [1746].log_data[7].valid := 1, [1746].log_data[8].valid := 1, [1746].log_data[9].valid := 1, [1746].log_data[10].valid := 1, [1746].log_data[11].valid := 1, [1746].log_data[12].valid := 1, [1746].log_data[13].valid := 1, [1746].log_data[14].valid := 1, [1746].log_data[15].valid := 1, [1746].log_data[16].valid := 1, [1746].log_data[17].valid := 1, [1746].log_data[18].valid := 1, [1746].log_data[19].valid := 1, [1746].time.Year := 2023, [1746].time.Month := 1, [1746].time.Day := 15, [1746].time.Hour := 17, [1746].time.Minute := 54, [1746].time.Second := 59, [1747].log_data[0].min := 1.0, [1747].log_data[0].max := 1.0, [1747].log_data[0].total := 300.0, [1747].log_data[0].time := 300.0, [1747].log_data[0].minminute := 55, [1747].log_data[0].maxminute := 55, [1747].log_data[0].valid := 1, [1747].log_data[1].valid := 1, [1747].log_data[2].valid := 1, [1747].log_data[3].valid := 1, [1747].log_data[4].valid := 1, [1747].log_data[5].valid := 1, [1747].log_data[6].valid := 1, [1747].log_data[7].valid := 1, [1747].log_data[8].valid := 1, [1747].log_data[9].valid := 1, [1747].log_data[10].valid := 1, [1747].log_data[11].valid := 1, [1747].log_data[12].valid := 1, [1747].log_data[13].valid := 1,
        [1747].log_data[14].valid := 1, [1747].log_data[15].valid := 1, [1747].log_data[16].valid := 1, [1747].log_data[17].valid := 1, [1747].log_data[18].valid := 1, [1747].log_data[19].valid := 1, [1747].time.Year := 2023, [1747].time.Month := 1, [1747].time.Day := 15, [1747].time.Hour := 17, [1747].time.Minute := 59, [1747].time.Second := 59, [1748].log_data[0].min := 1.0, [1748].log_data[0].max := 1.0, [1748].log_data[0].total := 300.0, [1748].log_data[0].time := 300.0, [1748].log_data[0].valid := 1, [1748].log_data[1].valid := 1, [1748].log_data[2].valid := 1, [1748].log_data[3].valid := 1, [1748].log_data[4].valid := 1, [1748].log_data[5].valid := 1, [1748].log_data[6].valid := 1, [1748].log_data[7].valid := 1, [1748].log_data[8].valid := 1, [1748].log_data[9].valid := 1, [1748].log_data[10].valid := 1, [1748].log_data[11].valid := 1, [1748].log_data[12].valid := 1, [1748].log_data[13].valid := 1, [1748].log_data[14].valid := 1, [1748].log_data[15].valid := 1, [1748].log_data[16].valid := 1, [1748].log_data[17].valid := 1, [1748].log_data[18].valid := 1, [1748].log_data[19].valid := 1, [1748].time.Year := 2023, [1748].time.Month := 1, [1748].time.Day := 15, [1748].time.Hour := 18, [1748].time.Minute := 4, [1748].time.Second := 59, [1749].log_data[0].min := 1.0, [1749].log_data[0].max := 1.0, [1749].log_data[0].total := 300.0, [1749].log_data[0].time := 300.0, [1749].log_data[0].minminute := 5, [1749].log_data[0].maxminute := 5, [1749].log_data[0].valid := 1, [1749].log_data[1].valid := 1, [1749].log_data[2].valid := 1, [1749].log_data[3].valid := 1, [1749].log_data[4].valid := 1, [1749].log_data[5].valid := 1, [1749].log_data[6].valid := 1, [1749].log_data[7].valid := 1, [1749].log_data[8].valid := 1, [1749].log_data[9].valid := 1, [1749].log_data[10].valid := 1, [1749].log_data[11].valid := 1,
        [1749].log_data[12].valid := 1, [1749].log_data[13].valid := 1, [1749].log_data[14].valid := 1, [1749].log_data[15].valid := 1, [1749].log_data[16].valid := 1, [1749].log_data[17].valid := 1, [1749].log_data[18].valid := 1, [1749].log_data[19].valid := 1, [1749].time.Year := 2023, [1749].time.Month := 1, [1749].time.Day := 15, [1749].time.Hour := 18, [1749].time.Minute := 9, [1749].time.Second := 59, [1750].log_data[0].min := 1.0, [1750].log_data[0].max := 1.0, [1750].log_data[0].total := 300.0, [1750].log_data[0].time := 300.0, [1750].log_data[0].minminute := 10, [1750].log_data[0].maxminute := 10, [1750].log_data[0].valid := 1, [1750].log_data[1].valid := 1, [1750].log_data[2].valid := 1, [1750].log_data[3].valid := 1, [1750].log_data[4].valid := 1, [1750].log_data[5].valid := 1, [1750].log_data[6].valid := 1, [1750].log_data[7].valid := 1, [1750].log_data[8].valid := 1, [1750].log_data[9].valid := 1, [1750].log_data[10].valid := 1, [1750].log_data[11].valid := 1, [1750].log_data[12].valid := 1, [1750].log_data[13].valid := 1, [1750].log_data[14].valid := 1, [1750].log_data[15].valid := 1, [1750].log_data[16].valid := 1, [1750].log_data[17].valid := 1, [1750].log_data[18].valid := 1, [1750].log_data[19].valid := 1, [1750].time.Year := 2023, [1750].time.Month := 1, [1750].time.Day := 15, [1750].time.Hour := 18, [1750].time.Minute := 14, [1750].time.Second := 59, [1751].log_data[0].min := 1.0, [1751].log_data[0].max := 1.0, [1751].log_data[0].total := 300.0, [1751].log_data[0].time := 300.0, [1751].log_data[0].minminute := 15, [1751].log_data[0].maxminute := 15, [1751].log_data[0].valid := 1, [1751].log_data[1].valid := 1, [1751].log_data[2].valid := 1, [1751].log_data[3].valid := 1, [1751].log_data[4].valid := 1, [1751].log_data[5].valid := 1, [1751].log_data[6].valid := 1, [1751].log_data[7].valid := 1,
        [1751].log_data[8].valid := 1, [1751].log_data[9].valid := 1, [1751].log_data[10].valid := 1, [1751].log_data[11].valid := 1, [1751].log_data[12].valid := 1, [1751].log_data[13].valid := 1, [1751].log_data[14].valid := 1, [1751].log_data[15].valid := 1, [1751].log_data[16].valid := 1, [1751].log_data[17].valid := 1, [1751].log_data[18].valid := 1, [1751].log_data[19].valid := 1, [1751].time.Year := 2023, [1751].time.Month := 1, [1751].time.Day := 15, [1751].time.Hour := 18, [1751].time.Minute := 19, [1751].time.Second := 59, [1752].log_data[0].min := 1.0, [1752].log_data[0].max := 1.0, [1752].log_data[0].total := 300.0, [1752].log_data[0].time := 300.0, [1752].log_data[0].minminute := 20, [1752].log_data[0].maxminute := 20, [1752].log_data[0].valid := 1, [1752].log_data[1].valid := 1, [1752].log_data[2].valid := 1, [1752].log_data[3].valid := 1, [1752].log_data[4].valid := 1, [1752].log_data[5].valid := 1, [1752].log_data[6].valid := 1, [1752].log_data[7].valid := 1, [1752].log_data[8].valid := 1, [1752].log_data[9].valid := 1, [1752].log_data[10].valid := 1, [1752].log_data[11].valid := 1, [1752].log_data[12].valid := 1, [1752].log_data[13].valid := 1, [1752].log_data[14].valid := 1, [1752].log_data[15].valid := 1, [1752].log_data[16].valid := 1, [1752].log_data[17].valid := 1, [1752].log_data[18].valid := 1, [1752].log_data[19].valid := 1, [1752].time.Year := 2023, [1752].time.Month := 1, [1752].time.Day := 15, [1752].time.Hour := 18, [1752].time.Minute := 24, [1752].time.Second := 59, [1753].log_data[0].min := 1.0, [1753].log_data[0].max := 1.0, [1753].log_data[0].total := 300.0, [1753].log_data[0].time := 300.0, [1753].log_data[0].minminute := 25, [1753].log_data[0].maxminute := 25, [1753].log_data[0].valid := 1, [1753].log_data[1].valid := 1, [1753].log_data[2].valid := 1, [1753].log_data[3].valid := 1,
        [1753].log_data[4].valid := 1, [1753].log_data[5].valid := 1, [1753].log_data[6].valid := 1, [1753].log_data[7].valid := 1, [1753].log_data[8].valid := 1, [1753].log_data[9].valid := 1, [1753].log_data[10].valid := 1, [1753].log_data[11].valid := 1, [1753].log_data[12].valid := 1, [1753].log_data[13].valid := 1, [1753].log_data[14].valid := 1, [1753].log_data[15].valid := 1, [1753].log_data[16].valid := 1, [1753].log_data[17].valid := 1, [1753].log_data[18].valid := 1, [1753].log_data[19].valid := 1, [1753].time.Year := 2023, [1753].time.Month := 1, [1753].time.Day := 15, [1753].time.Hour := 18, [1753].time.Minute := 29, [1753].time.Second := 59, [1754].log_data[0].min := 1.0, [1754].log_data[0].max := 1.0, [1754].log_data[0].total := 300.0, [1754].log_data[0].time := 300.0, [1754].log_data[0].minminute := 30, [1754].log_data[0].maxminute := 30, [1754].log_data[0].valid := 1, [1754].log_data[1].valid := 1, [1754].log_data[2].valid := 1, [1754].log_data[3].valid := 1, [1754].log_data[4].valid := 1, [1754].log_data[5].valid := 1, [1754].log_data[6].valid := 1, [1754].log_data[7].valid := 1, [1754].log_data[8].valid := 1, [1754].log_data[9].valid := 1, [1754].log_data[10].valid := 1, [1754].log_data[11].valid := 1, [1754].log_data[12].valid := 1, [1754].log_data[13].valid := 1, [1754].log_data[14].valid := 1, [1754].log_data[15].valid := 1, [1754].log_data[16].valid := 1, [1754].log_data[17].valid := 1, [1754].log_data[18].valid := 1, [1754].log_data[19].valid := 1, [1754].time.Year := 2023, [1754].time.Month := 1, [1754].time.Day := 15, [1754].time.Hour := 18, [1754].time.Minute := 34, [1754].time.Second := 59, [1755].log_data[0].min := 1.0, [1755].log_data[0].max := 1.0, [1755].log_data[0].total := 300.0, [1755].log_data[0].time := 300.0, [1755].log_data[0].minminute := 35, [1755].log_data[0].maxminute := 35,
        [1755].log_data[0].valid := 1, [1755].log_data[1].valid := 1, [1755].log_data[2].valid := 1, [1755].log_data[3].valid := 1, [1755].log_data[4].valid := 1, [1755].log_data[5].valid := 1, [1755].log_data[6].valid := 1, [1755].log_data[7].valid := 1, [1755].log_data[8].valid := 1, [1755].log_data[9].valid := 1, [1755].log_data[10].valid := 1, [1755].log_data[11].valid := 1, [1755].log_data[12].valid := 1, [1755].log_data[13].valid := 1, [1755].log_data[14].valid := 1, [1755].log_data[15].valid := 1, [1755].log_data[16].valid := 1, [1755].log_data[17].valid := 1, [1755].log_data[18].valid := 1, [1755].log_data[19].valid := 1, [1755].time.Year := 2023, [1755].time.Month := 1, [1755].time.Day := 15, [1755].time.Hour := 18, [1755].time.Minute := 39, [1755].time.Second := 59, [1756].log_data[0].min := 1.0, [1756].log_data[0].max := 1.0, [1756].log_data[0].total := 300.0, [1756].log_data[0].time := 300.0, [1756].log_data[0].minminute := 40, [1756].log_data[0].maxminute := 40, [1756].log_data[0].valid := 1, [1756].log_data[1].valid := 1, [1756].log_data[2].valid := 1, [1756].log_data[3].valid := 1, [1756].log_data[4].valid := 1, [1756].log_data[5].valid := 1, [1756].log_data[6].valid := 1, [1756].log_data[7].valid := 1, [1756].log_data[8].valid := 1, [1756].log_data[9].valid := 1, [1756].log_data[10].valid := 1, [1756].log_data[11].valid := 1, [1756].log_data[12].valid := 1, [1756].log_data[13].valid := 1, [1756].log_data[14].valid := 1, [1756].log_data[15].valid := 1, [1756].log_data[16].valid := 1, [1756].log_data[17].valid := 1, [1756].log_data[18].valid := 1, [1756].log_data[19].valid := 1, [1756].time.Year := 2023, [1756].time.Month := 1, [1756].time.Day := 15, [1756].time.Hour := 18, [1756].time.Minute := 44, [1756].time.Second := 59, [1757].log_data[0].min := 1.0, [1757].log_data[0].max := 1.0,
        [1757].log_data[0].total := 300.0, [1757].log_data[0].time := 300.0, [1757].log_data[0].minminute := 45, [1757].log_data[0].maxminute := 45, [1757].log_data[0].valid := 1, [1757].log_data[1].valid := 1, [1757].log_data[2].valid := 1, [1757].log_data[3].valid := 1, [1757].log_data[4].valid := 1, [1757].log_data[5].valid := 1, [1757].log_data[6].valid := 1, [1757].log_data[7].valid := 1, [1757].log_data[8].valid := 1, [1757].log_data[9].valid := 1, [1757].log_data[10].valid := 1, [1757].log_data[11].valid := 1, [1757].log_data[12].valid := 1, [1757].log_data[13].valid := 1, [1757].log_data[14].valid := 1, [1757].log_data[15].valid := 1, [1757].log_data[16].valid := 1, [1757].log_data[17].valid := 1, [1757].log_data[18].valid := 1, [1757].log_data[19].valid := 1, [1757].time.Year := 2023, [1757].time.Month := 1, [1757].time.Day := 15, [1757].time.Hour := 18, [1757].time.Minute := 49, [1757].time.Second := 59, [1758].log_data[0].min := 1.0, [1758].log_data[0].max := 1.0, [1758].log_data[0].total := 300.0, [1758].log_data[0].time := 300.0, [1758].log_data[0].minminute := 50, [1758].log_data[0].maxminute := 50, [1758].log_data[0].valid := 1, [1758].log_data[1].valid := 1, [1758].log_data[2].valid := 1, [1758].log_data[3].valid := 1, [1758].log_data[4].valid := 1, [1758].log_data[5].valid := 1, [1758].log_data[6].valid := 1, [1758].log_data[7].valid := 1, [1758].log_data[8].valid := 1, [1758].log_data[9].valid := 1, [1758].log_data[10].valid := 1, [1758].log_data[11].valid := 1, [1758].log_data[12].valid := 1, [1758].log_data[13].valid := 1, [1758].log_data[14].valid := 1, [1758].log_data[15].valid := 1, [1758].log_data[16].valid := 1, [1758].log_data[17].valid := 1, [1758].log_data[18].valid := 1, [1758].log_data[19].valid := 1, [1758].time.Year := 2023, [1758].time.Month := 1, [1758].time.Day := 15, [1758].time.Hour := 18,
        [1758].time.Minute := 54, [1758].time.Second := 59, [1759].log_data[0].min := 1.0, [1759].log_data[0].max := 1.0, [1759].log_data[0].total := 300.0, [1759].log_data[0].time := 300.0, [1759].log_data[0].minminute := 55, [1759].log_data[0].maxminute := 55, [1759].log_data[0].valid := 1, [1759].log_data[1].valid := 1, [1759].log_data[2].valid := 1, [1759].log_data[3].valid := 1, [1759].log_data[4].valid := 1, [1759].log_data[5].valid := 1, [1759].log_data[6].valid := 1, [1759].log_data[7].valid := 1, [1759].log_data[8].valid := 1, [1759].log_data[9].valid := 1, [1759].log_data[10].valid := 1, [1759].log_data[11].valid := 1, [1759].log_data[12].valid := 1, [1759].log_data[13].valid := 1, [1759].log_data[14].valid := 1, [1759].log_data[15].valid := 1, [1759].log_data[16].valid := 1, [1759].log_data[17].valid := 1, [1759].log_data[18].valid := 1, [1759].log_data[19].valid := 1, [1759].time.Year := 2023, [1759].time.Month := 1, [1759].time.Day := 15, [1759].time.Hour := 18, [1759].time.Minute := 59, [1759].time.Second := 59, [1760].log_data[0].min := 1.0, [1760].log_data[0].max := 1.0, [1760].log_data[0].total := 300.0, [1760].log_data[0].time := 300.0, [1760].log_data[0].valid := 1, [1760].log_data[1].valid := 1, [1760].log_data[2].valid := 1, [1760].log_data[3].valid := 1, [1760].log_data[4].valid := 1, [1760].log_data[5].valid := 1, [1760].log_data[6].valid := 1, [1760].log_data[7].valid := 1, [1760].log_data[8].valid := 1, [1760].log_data[9].valid := 1, [1760].log_data[10].valid := 1, [1760].log_data[11].valid := 1, [1760].log_data[12].valid := 1, [1760].log_data[13].valid := 1, [1760].log_data[14].valid := 1, [1760].log_data[15].valid := 1, [1760].log_data[16].valid := 1, [1760].log_data[17].valid := 1, [1760].log_data[18].valid := 1, [1760].log_data[19].valid := 1, [1760].time.Year := 2023, [1760].time.Month := 1,
        [1760].time.Day := 15, [1760].time.Hour := 19, [1760].time.Minute := 4, [1760].time.Second := 59, [1761].log_data[0].min := 1.0, [1761].log_data[0].max := 1.0, [1761].log_data[0].total := 300.0, [1761].log_data[0].time := 300.0, [1761].log_data[0].minminute := 5, [1761].log_data[0].maxminute := 5, [1761].log_data[0].valid := 1, [1761].log_data[1].valid := 1, [1761].log_data[2].valid := 1, [1761].log_data[3].valid := 1, [1761].log_data[4].valid := 1, [1761].log_data[5].valid := 1, [1761].log_data[6].valid := 1, [1761].log_data[7].valid := 1, [1761].log_data[8].valid := 1, [1761].log_data[9].valid := 1, [1761].log_data[10].valid := 1, [1761].log_data[11].valid := 1, [1761].log_data[12].valid := 1, [1761].log_data[13].valid := 1, [1761].log_data[14].valid := 1, [1761].log_data[15].valid := 1, [1761].log_data[16].valid := 1, [1761].log_data[17].valid := 1, [1761].log_data[18].valid := 1, [1761].log_data[19].valid := 1, [1761].time.Year := 2023, [1761].time.Month := 1, [1761].time.Day := 15, [1761].time.Hour := 19, [1761].time.Minute := 9, [1761].time.Second := 59, [1762].log_data[0].min := 1.0, [1762].log_data[0].max := 1.0, [1762].log_data[0].total := 300.0, [1762].log_data[0].time := 300.0, [1762].log_data[0].minminute := 10, [1762].log_data[0].maxminute := 10, [1762].log_data[0].valid := 1, [1762].log_data[1].valid := 1, [1762].log_data[2].valid := 1, [1762].log_data[3].valid := 1, [1762].log_data[4].valid := 1, [1762].log_data[5].valid := 1, [1762].log_data[6].valid := 1, [1762].log_data[7].valid := 1, [1762].log_data[8].valid := 1, [1762].log_data[9].valid := 1, [1762].log_data[10].valid := 1, [1762].log_data[11].valid := 1, [1762].log_data[12].valid := 1, [1762].log_data[13].valid := 1, [1762].log_data[14].valid := 1, [1762].log_data[15].valid := 1, [1762].log_data[16].valid := 1, [1762].log_data[17].valid := 1,
        [1762].log_data[18].valid := 1, [1762].log_data[19].valid := 1, [1762].time.Year := 2023, [1762].time.Month := 1, [1762].time.Day := 15, [1762].time.Hour := 19, [1762].time.Minute := 14, [1762].time.Second := 59, [1763].log_data[0].min := 1.0, [1763].log_data[0].max := 1.0, [1763].log_data[0].total := 300.0, [1763].log_data[0].time := 300.0, [1763].log_data[0].minminute := 15, [1763].log_data[0].maxminute := 15, [1763].log_data[0].valid := 1, [1763].log_data[1].valid := 1, [1763].log_data[2].valid := 1, [1763].log_data[3].valid := 1, [1763].log_data[4].valid := 1, [1763].log_data[5].valid := 1, [1763].log_data[6].valid := 1, [1763].log_data[7].valid := 1, [1763].log_data[8].valid := 1, [1763].log_data[9].valid := 1, [1763].log_data[10].valid := 1, [1763].log_data[11].valid := 1, [1763].log_data[12].valid := 1, [1763].log_data[13].valid := 1, [1763].log_data[14].valid := 1, [1763].log_data[15].valid := 1, [1763].log_data[16].valid := 1, [1763].log_data[17].valid := 1, [1763].log_data[18].valid := 1, [1763].log_data[19].valid := 1, [1763].time.Year := 2023, [1763].time.Month := 1, [1763].time.Day := 15, [1763].time.Hour := 19, [1763].time.Minute := 19, [1763].time.Second := 59, [1764].log_data[0].min := 1.0, [1764].log_data[0].max := 1.0, [1764].log_data[0].total := 300.0, [1764].log_data[0].time := 300.0, [1764].log_data[0].minminute := 20, [1764].log_data[0].maxminute := 20, [1764].log_data[0].valid := 1, [1764].log_data[1].valid := 1, [1764].log_data[2].valid := 1, [1764].log_data[3].valid := 1, [1764].log_data[4].valid := 1, [1764].log_data[5].valid := 1, [1764].log_data[6].valid := 1, [1764].log_data[7].valid := 1, [1764].log_data[8].valid := 1, [1764].log_data[9].valid := 1, [1764].log_data[10].valid := 1, [1764].log_data[11].valid := 1, [1764].log_data[12].valid := 1, [1764].log_data[13].valid := 1,
        [1764].log_data[14].valid := 1, [1764].log_data[15].valid := 1, [1764].log_data[16].valid := 1, [1764].log_data[17].valid := 1, [1764].log_data[18].valid := 1, [1764].log_data[19].valid := 1, [1764].time.Year := 2023, [1764].time.Month := 1, [1764].time.Day := 15, [1764].time.Hour := 19, [1764].time.Minute := 24, [1764].time.Second := 59, [1765].log_data[0].min := 1.0, [1765].log_data[0].max := 1.0, [1765].log_data[0].total := 300.0, [1765].log_data[0].time := 300.0, [1765].log_data[0].minminute := 25, [1765].log_data[0].maxminute := 25, [1765].log_data[0].valid := 1, [1765].log_data[1].valid := 1, [1765].log_data[2].valid := 1, [1765].log_data[3].valid := 1, [1765].log_data[4].valid := 1, [1765].log_data[5].valid := 1, [1765].log_data[6].valid := 1, [1765].log_data[7].valid := 1, [1765].log_data[8].valid := 1, [1765].log_data[9].valid := 1, [1765].log_data[10].valid := 1, [1765].log_data[11].valid := 1, [1765].log_data[12].valid := 1, [1765].log_data[13].valid := 1, [1765].log_data[14].valid := 1, [1765].log_data[15].valid := 1, [1765].log_data[16].valid := 1, [1765].log_data[17].valid := 1, [1765].log_data[18].valid := 1, [1765].log_data[19].valid := 1, [1765].time.Year := 2023, [1765].time.Month := 1, [1765].time.Day := 15, [1765].time.Hour := 19, [1765].time.Minute := 29, [1765].time.Second := 59, [1766].log_data[0].min := 1.0, [1766].log_data[0].max := 1.0, [1766].log_data[0].total := 300.0, [1766].log_data[0].time := 300.0, [1766].log_data[0].minminute := 30, [1766].log_data[0].maxminute := 30, [1766].log_data[0].valid := 1, [1766].log_data[1].valid := 1, [1766].log_data[2].valid := 1, [1766].log_data[3].valid := 1, [1766].log_data[4].valid := 1, [1766].log_data[5].valid := 1, [1766].log_data[6].valid := 1, [1766].log_data[7].valid := 1, [1766].log_data[8].valid := 1, [1766].log_data[9].valid := 1,
        [1766].log_data[10].valid := 1, [1766].log_data[11].valid := 1, [1766].log_data[12].valid := 1, [1766].log_data[13].valid := 1, [1766].log_data[14].valid := 1, [1766].log_data[15].valid := 1, [1766].log_data[16].valid := 1, [1766].log_data[17].valid := 1, [1766].log_data[18].valid := 1, [1766].log_data[19].valid := 1, [1766].time.Year := 2023, [1766].time.Month := 1, [1766].time.Day := 15, [1766].time.Hour := 19, [1766].time.Minute := 34, [1766].time.Second := 59, [1767].log_data[0].min := 1.0, [1767].log_data[0].max := 1.0, [1767].log_data[0].total := 300.0, [1767].log_data[0].time := 300.0, [1767].log_data[0].minminute := 35, [1767].log_data[0].maxminute := 35, [1767].log_data[0].valid := 1, [1767].log_data[1].valid := 1, [1767].log_data[2].valid := 1, [1767].log_data[3].valid := 1, [1767].log_data[4].valid := 1, [1767].log_data[5].valid := 1, [1767].log_data[6].valid := 1, [1767].log_data[7].valid := 1, [1767].log_data[8].valid := 1, [1767].log_data[9].valid := 1, [1767].log_data[10].valid := 1, [1767].log_data[11].valid := 1, [1767].log_data[12].valid := 1, [1767].log_data[13].valid := 1, [1767].log_data[14].valid := 1, [1767].log_data[15].valid := 1, [1767].log_data[16].valid := 1, [1767].log_data[17].valid := 1, [1767].log_data[18].valid := 1, [1767].log_data[19].valid := 1, [1767].time.Year := 2023, [1767].time.Month := 1, [1767].time.Day := 15, [1767].time.Hour := 19, [1767].time.Minute := 39, [1767].time.Second := 59, [1768].log_data[0].min := 1.0, [1768].log_data[0].max := 1.0, [1768].log_data[0].total := 300.0, [1768].log_data[0].time := 300.0, [1768].log_data[0].minminute := 40, [1768].log_data[0].maxminute := 40, [1768].log_data[0].valid := 1, [1768].log_data[1].valid := 1, [1768].log_data[2].valid := 1, [1768].log_data[3].valid := 1, [1768].log_data[4].valid := 1, [1768].log_data[5].valid := 1,
        [1768].log_data[6].valid := 1, [1768].log_data[7].valid := 1, [1768].log_data[8].valid := 1, [1768].log_data[9].valid := 1, [1768].log_data[10].valid := 1, [1768].log_data[11].valid := 1, [1768].log_data[12].valid := 1, [1768].log_data[13].valid := 1, [1768].log_data[14].valid := 1, [1768].log_data[15].valid := 1, [1768].log_data[16].valid := 1, [1768].log_data[17].valid := 1, [1768].log_data[18].valid := 1, [1768].log_data[19].valid := 1, [1768].time.Year := 2023, [1768].time.Month := 1, [1768].time.Day := 15, [1768].time.Hour := 19, [1768].time.Minute := 44, [1768].time.Second := 59, [1769].log_data[0].min := 1.0, [1769].log_data[0].max := 1.0, [1769].log_data[0].total := 300.0, [1769].log_data[0].time := 300.0, [1769].log_data[0].minminute := 45, [1769].log_data[0].maxminute := 45, [1769].log_data[0].valid := 1, [1769].log_data[1].valid := 1, [1769].log_data[2].valid := 1, [1769].log_data[3].valid := 1, [1769].log_data[4].valid := 1, [1769].log_data[5].valid := 1, [1769].log_data[6].valid := 1, [1769].log_data[7].valid := 1, [1769].log_data[8].valid := 1, [1769].log_data[9].valid := 1, [1769].log_data[10].valid := 1, [1769].log_data[11].valid := 1, [1769].log_data[12].valid := 1, [1769].log_data[13].valid := 1, [1769].log_data[14].valid := 1, [1769].log_data[15].valid := 1, [1769].log_data[16].valid := 1, [1769].log_data[17].valid := 1, [1769].log_data[18].valid := 1, [1769].log_data[19].valid := 1, [1769].time.Year := 2023, [1769].time.Month := 1, [1769].time.Day := 15, [1769].time.Hour := 19, [1769].time.Minute := 49, [1769].time.Second := 59, [1770].log_data[0].min := 1.0, [1770].log_data[0].max := 1.0, [1770].log_data[0].total := 300.0, [1770].log_data[0].time := 300.0, [1770].log_data[0].minminute := 50, [1770].log_data[0].maxminute := 50, [1770].log_data[0].valid := 1, [1770].log_data[1].valid := 1,
        [1770].log_data[2].valid := 1, [1770].log_data[3].valid := 1, [1770].log_data[4].valid := 1, [1770].log_data[5].valid := 1, [1770].log_data[6].valid := 1, [1770].log_data[7].valid := 1, [1770].log_data[8].valid := 1, [1770].log_data[9].valid := 1, [1770].log_data[10].valid := 1, [1770].log_data[11].valid := 1, [1770].log_data[12].valid := 1, [1770].log_data[13].valid := 1, [1770].log_data[14].valid := 1, [1770].log_data[15].valid := 1, [1770].log_data[16].valid := 1, [1770].log_data[17].valid := 1, [1770].log_data[18].valid := 1, [1770].log_data[19].valid := 1, [1770].time.Year := 2023, [1770].time.Month := 1, [1770].time.Day := 15, [1770].time.Hour := 19, [1770].time.Minute := 54, [1770].time.Second := 59, [1771].log_data[0].min := 1.0, [1771].log_data[0].max := 1.0, [1771].log_data[0].total := 300.0, [1771].log_data[0].time := 300.0, [1771].log_data[0].minminute := 55, [1771].log_data[0].maxminute := 55, [1771].log_data[0].valid := 1, [1771].log_data[1].valid := 1, [1771].log_data[2].valid := 1, [1771].log_data[3].valid := 1, [1771].log_data[4].valid := 1, [1771].log_data[5].valid := 1, [1771].log_data[6].valid := 1, [1771].log_data[7].valid := 1, [1771].log_data[8].valid := 1, [1771].log_data[9].valid := 1, [1771].log_data[10].valid := 1, [1771].log_data[11].valid := 1, [1771].log_data[12].valid := 1, [1771].log_data[13].valid := 1, [1771].log_data[14].valid := 1, [1771].log_data[15].valid := 1, [1771].log_data[16].valid := 1, [1771].log_data[17].valid := 1, [1771].log_data[18].valid := 1, [1771].log_data[19].valid := 1, [1771].time.Year := 2023, [1771].time.Month := 1, [1771].time.Day := 15, [1771].time.Hour := 19, [1771].time.Minute := 59, [1771].time.Second := 59, [1772].log_data[0].min := 1.0, [1772].log_data[0].max := 1.0, [1772].log_data[0].total := 300.0, [1772].log_data[0].time := 300.0,
        [1772].log_data[0].valid := 1, [1772].log_data[1].valid := 1, [1772].log_data[2].valid := 1, [1772].log_data[3].valid := 1, [1772].log_data[4].valid := 1, [1772].log_data[5].valid := 1, [1772].log_data[6].valid := 1, [1772].log_data[7].valid := 1, [1772].log_data[8].valid := 1, [1772].log_data[9].valid := 1, [1772].log_data[10].valid := 1, [1772].log_data[11].valid := 1, [1772].log_data[12].valid := 1, [1772].log_data[13].valid := 1, [1772].log_data[14].valid := 1, [1772].log_data[15].valid := 1, [1772].log_data[16].valid := 1, [1772].log_data[17].valid := 1, [1772].log_data[18].valid := 1, [1772].log_data[19].valid := 1, [1772].time.Year := 2023, [1772].time.Month := 1, [1772].time.Day := 15, [1772].time.Hour := 20, [1772].time.Minute := 4, [1772].time.Second := 59, [1773].log_data[0].min := 1.0, [1773].log_data[0].max := 1.0, [1773].log_data[0].total := 300.0, [1773].log_data[0].time := 300.0, [1773].log_data[0].minminute := 5, [1773].log_data[0].maxminute := 5, [1773].log_data[0].valid := 1, [1773].log_data[1].valid := 1, [1773].log_data[2].valid := 1, [1773].log_data[3].valid := 1, [1773].log_data[4].valid := 1, [1773].log_data[5].valid := 1, [1773].log_data[6].valid := 1, [1773].log_data[7].valid := 1, [1773].log_data[8].valid := 1, [1773].log_data[9].valid := 1, [1773].log_data[10].valid := 1, [1773].log_data[11].valid := 1, [1773].log_data[12].valid := 1, [1773].log_data[13].valid := 1, [1773].log_data[14].valid := 1, [1773].log_data[15].valid := 1, [1773].log_data[16].valid := 1, [1773].log_data[17].valid := 1, [1773].log_data[18].valid := 1, [1773].log_data[19].valid := 1, [1773].time.Year := 2023, [1773].time.Month := 1, [1773].time.Day := 15, [1773].time.Hour := 20, [1773].time.Minute := 9, [1773].time.Second := 59, [1774].log_data[0].min := 1.0, [1774].log_data[0].max := 1.0,
        [1774].log_data[0].total := 300.0, [1774].log_data[0].time := 300.0, [1774].log_data[0].minminute := 10, [1774].log_data[0].maxminute := 10, [1774].log_data[0].valid := 1, [1774].log_data[1].valid := 1, [1774].log_data[2].valid := 1, [1774].log_data[3].valid := 1, [1774].log_data[4].valid := 1, [1774].log_data[5].valid := 1, [1774].log_data[6].valid := 1, [1774].log_data[7].valid := 1, [1774].log_data[8].valid := 1, [1774].log_data[9].valid := 1, [1774].log_data[10].valid := 1, [1774].log_data[11].valid := 1, [1774].log_data[12].valid := 1, [1774].log_data[13].valid := 1, [1774].log_data[14].valid := 1, [1774].log_data[15].valid := 1, [1774].log_data[16].valid := 1, [1774].log_data[17].valid := 1, [1774].log_data[18].valid := 1, [1774].log_data[19].valid := 1, [1774].time.Year := 2023, [1774].time.Month := 1, [1774].time.Day := 15, [1774].time.Hour := 20, [1774].time.Minute := 14, [1774].time.Second := 59, [1775].log_data[0].min := 1.0, [1775].log_data[0].max := 1.0, [1775].log_data[0].total := 300.0, [1775].log_data[0].time := 300.0, [1775].log_data[0].minminute := 15, [1775].log_data[0].maxminute := 15, [1775].log_data[0].valid := 1, [1775].log_data[1].valid := 1, [1775].log_data[2].valid := 1, [1775].log_data[3].valid := 1, [1775].log_data[4].valid := 1, [1775].log_data[5].valid := 1, [1775].log_data[6].valid := 1, [1775].log_data[7].valid := 1, [1775].log_data[8].valid := 1, [1775].log_data[9].valid := 1, [1775].log_data[10].valid := 1, [1775].log_data[11].valid := 1, [1775].log_data[12].valid := 1, [1775].log_data[13].valid := 1, [1775].log_data[14].valid := 1, [1775].log_data[15].valid := 1, [1775].log_data[16].valid := 1, [1775].log_data[17].valid := 1, [1775].log_data[18].valid := 1, [1775].log_data[19].valid := 1, [1775].time.Year := 2023, [1775].time.Month := 1, [1775].time.Day := 15, [1775].time.Hour := 20,
        [1775].time.Minute := 19, [1775].time.Second := 59, [1776].log_data[0].min := 1.0, [1776].log_data[0].max := 1.0, [1776].log_data[0].total := 300.0, [1776].log_data[0].time := 300.0, [1776].log_data[0].minminute := 20, [1776].log_data[0].maxminute := 20, [1776].log_data[0].valid := 1, [1776].log_data[1].valid := 1, [1776].log_data[2].valid := 1, [1776].log_data[3].valid := 1, [1776].log_data[4].valid := 1, [1776].log_data[5].valid := 1, [1776].log_data[6].valid := 1, [1776].log_data[7].valid := 1, [1776].log_data[8].valid := 1, [1776].log_data[9].valid := 1, [1776].log_data[10].valid := 1, [1776].log_data[11].valid := 1, [1776].log_data[12].valid := 1, [1776].log_data[13].valid := 1, [1776].log_data[14].valid := 1, [1776].log_data[15].valid := 1, [1776].log_data[16].valid := 1, [1776].log_data[17].valid := 1, [1776].log_data[18].valid := 1, [1776].log_data[19].valid := 1, [1776].time.Year := 2023, [1776].time.Month := 1, [1776].time.Day := 15, [1776].time.Hour := 20, [1776].time.Minute := 24, [1776].time.Second := 59, [1777].log_data[0].min := 1.0, [1777].log_data[0].max := 1.0, [1777].log_data[0].total := 300.0, [1777].log_data[0].time := 300.0, [1777].log_data[0].minminute := 25, [1777].log_data[0].maxminute := 25, [1777].log_data[0].valid := 1, [1777].log_data[1].valid := 1, [1777].log_data[2].valid := 1, [1777].log_data[3].valid := 1, [1777].log_data[4].valid := 1, [1777].log_data[5].valid := 1, [1777].log_data[6].valid := 1, [1777].log_data[7].valid := 1, [1777].log_data[8].valid := 1, [1777].log_data[9].valid := 1, [1777].log_data[10].valid := 1, [1777].log_data[11].valid := 1, [1777].log_data[12].valid := 1, [1777].log_data[13].valid := 1, [1777].log_data[14].valid := 1, [1777].log_data[15].valid := 1, [1777].log_data[16].valid := 1, [1777].log_data[17].valid := 1, [1777].log_data[18].valid := 1, [1777].log_data[19].valid := 1,
        [1777].time.Year := 2023, [1777].time.Month := 1, [1777].time.Day := 15, [1777].time.Hour := 20, [1777].time.Minute := 29, [1777].time.Second := 59, [1778].log_data[0].min := 1.0, [1778].log_data[0].max := 1.0, [1778].log_data[0].total := 300.0, [1778].log_data[0].time := 300.0, [1778].log_data[0].minminute := 30, [1778].log_data[0].maxminute := 30, [1778].log_data[0].valid := 1, [1778].log_data[1].valid := 1, [1778].log_data[2].valid := 1, [1778].log_data[3].valid := 1, [1778].log_data[4].valid := 1, [1778].log_data[5].valid := 1, [1778].log_data[6].valid := 1, [1778].log_data[7].valid := 1, [1778].log_data[8].valid := 1, [1778].log_data[9].valid := 1, [1778].log_data[10].valid := 1, [1778].log_data[11].valid := 1, [1778].log_data[12].valid := 1, [1778].log_data[13].valid := 1, [1778].log_data[14].valid := 1, [1778].log_data[15].valid := 1, [1778].log_data[16].valid := 1, [1778].log_data[17].valid := 1, [1778].log_data[18].valid := 1, [1778].log_data[19].valid := 1, [1778].time.Year := 2023, [1778].time.Month := 1, [1778].time.Day := 15, [1778].time.Hour := 20, [1778].time.Minute := 34, [1778].time.Second := 59, [1779].log_data[0].min := 1.0, [1779].log_data[0].max := 1.0, [1779].log_data[0].total := 300.0, [1779].log_data[0].time := 300.0, [1779].log_data[0].minminute := 35, [1779].log_data[0].maxminute := 35, [1779].log_data[0].valid := 1, [1779].log_data[1].valid := 1, [1779].log_data[2].valid := 1, [1779].log_data[3].valid := 1, [1779].log_data[4].valid := 1, [1779].log_data[5].valid := 1, [1779].log_data[6].valid := 1, [1779].log_data[7].valid := 1, [1779].log_data[8].valid := 1, [1779].log_data[9].valid := 1, [1779].log_data[10].valid := 1, [1779].log_data[11].valid := 1, [1779].log_data[12].valid := 1, [1779].log_data[13].valid := 1, [1779].log_data[14].valid := 1, [1779].log_data[15].valid := 1,
        [1779].log_data[16].valid := 1, [1779].log_data[17].valid := 1, [1779].log_data[18].valid := 1, [1779].log_data[19].valid := 1, [1779].time.Year := 2023, [1779].time.Month := 1, [1779].time.Day := 15, [1779].time.Hour := 20, [1779].time.Minute := 39, [1779].time.Second := 59, [1780].log_data[0].min := 1.0, [1780].log_data[0].max := 1.0, [1780].log_data[0].total := 300.0, [1780].log_data[0].time := 300.0, [1780].log_data[0].minminute := 40, [1780].log_data[0].maxminute := 40, [1780].log_data[0].valid := 1, [1780].log_data[1].valid := 1, [1780].log_data[2].valid := 1, [1780].log_data[3].valid := 1, [1780].log_data[4].valid := 1, [1780].log_data[5].valid := 1, [1780].log_data[6].valid := 1, [1780].log_data[7].valid := 1, [1780].log_data[8].valid := 1, [1780].log_data[9].valid := 1, [1780].log_data[10].valid := 1, [1780].log_data[11].valid := 1, [1780].log_data[12].valid := 1, [1780].log_data[13].valid := 1, [1780].log_data[14].valid := 1, [1780].log_data[15].valid := 1, [1780].log_data[16].valid := 1, [1780].log_data[17].valid := 1, [1780].log_data[18].valid := 1, [1780].log_data[19].valid := 1, [1780].time.Year := 2023, [1780].time.Month := 1, [1780].time.Day := 15, [1780].time.Hour := 20, [1780].time.Minute := 44, [1780].time.Second := 59, [1781].log_data[0].min := 1.0, [1781].log_data[0].max := 1.0, [1781].log_data[0].total := 300.0, [1781].log_data[0].time := 300.0, [1781].log_data[0].minminute := 45, [1781].log_data[0].maxminute := 45, [1781].log_data[0].valid := 1, [1781].log_data[1].valid := 1, [1781].log_data[2].valid := 1, [1781].log_data[3].valid := 1, [1781].log_data[4].valid := 1, [1781].log_data[5].valid := 1, [1781].log_data[6].valid := 1, [1781].log_data[7].valid := 1, [1781].log_data[8].valid := 1, [1781].log_data[9].valid := 1, [1781].log_data[10].valid := 1, [1781].log_data[11].valid := 1,
        [1781].log_data[12].valid := 1, [1781].log_data[13].valid := 1, [1781].log_data[14].valid := 1, [1781].log_data[15].valid := 1, [1781].log_data[16].valid := 1, [1781].log_data[17].valid := 1, [1781].log_data[18].valid := 1, [1781].log_data[19].valid := 1, [1781].time.Year := 2023, [1781].time.Month := 1, [1781].time.Day := 15, [1781].time.Hour := 20, [1781].time.Minute := 49, [1781].time.Second := 59, [1782].log_data[0].min := 1.0, [1782].log_data[0].max := 1.0, [1782].log_data[0].total := 300.0, [1782].log_data[0].time := 300.0, [1782].log_data[0].minminute := 50, [1782].log_data[0].maxminute := 50, [1782].log_data[0].valid := 1, [1782].log_data[1].valid := 1, [1782].log_data[2].valid := 1, [1782].log_data[3].valid := 1, [1782].log_data[4].valid := 1, [1782].log_data[5].valid := 1, [1782].log_data[6].valid := 1, [1782].log_data[7].valid := 1, [1782].log_data[8].valid := 1, [1782].log_data[9].valid := 1, [1782].log_data[10].valid := 1, [1782].log_data[11].valid := 1, [1782].log_data[12].valid := 1, [1782].log_data[13].valid := 1, [1782].log_data[14].valid := 1, [1782].log_data[15].valid := 1, [1782].log_data[16].valid := 1, [1782].log_data[17].valid := 1, [1782].log_data[18].valid := 1, [1782].log_data[19].valid := 1, [1782].time.Year := 2023, [1782].time.Month := 1, [1782].time.Day := 15, [1782].time.Hour := 20, [1782].time.Minute := 54, [1782].time.Second := 59, [1783].log_data[0].min := 1.0, [1783].log_data[0].max := 1.0, [1783].log_data[0].total := 300.0, [1783].log_data[0].time := 300.0, [1783].log_data[0].minminute := 55, [1783].log_data[0].maxminute := 55, [1783].log_data[0].valid := 1, [1783].log_data[1].valid := 1, [1783].log_data[2].valid := 1, [1783].log_data[3].valid := 1, [1783].log_data[4].valid := 1, [1783].log_data[5].valid := 1, [1783].log_data[6].valid := 1, [1783].log_data[7].valid := 1,
        [1783].log_data[8].valid := 1, [1783].log_data[9].valid := 1, [1783].log_data[10].valid := 1, [1783].log_data[11].valid := 1, [1783].log_data[12].valid := 1, [1783].log_data[13].valid := 1, [1783].log_data[14].valid := 1, [1783].log_data[15].valid := 1, [1783].log_data[16].valid := 1, [1783].log_data[17].valid := 1, [1783].log_data[18].valid := 1, [1783].log_data[19].valid := 1, [1783].time.Year := 2023, [1783].time.Month := 1, [1783].time.Day := 15, [1783].time.Hour := 20, [1783].time.Minute := 59, [1783].time.Second := 59, [1784].log_data[0].min := 1.0, [1784].log_data[0].max := 1.0, [1784].log_data[0].total := 300.0, [1784].log_data[0].time := 300.0, [1784].log_data[0].valid := 1, [1784].log_data[1].valid := 1, [1784].log_data[2].valid := 1, [1784].log_data[3].valid := 1, [1784].log_data[4].valid := 1, [1784].log_data[5].valid := 1, [1784].log_data[6].valid := 1, [1784].log_data[7].valid := 1, [1784].log_data[8].valid := 1, [1784].log_data[9].valid := 1, [1784].log_data[10].valid := 1, [1784].log_data[11].valid := 1, [1784].log_data[12].valid := 1, [1784].log_data[13].valid := 1, [1784].log_data[14].valid := 1, [1784].log_data[15].valid := 1, [1784].log_data[16].valid := 1, [1784].log_data[17].valid := 1, [1784].log_data[18].valid := 1, [1784].log_data[19].valid := 1, [1784].time.Year := 2023, [1784].time.Month := 1, [1784].time.Day := 15, [1784].time.Hour := 21, [1784].time.Minute := 4, [1784].time.Second := 59, [1785].log_data[0].min := 1.0, [1785].log_data[0].max := 1.0, [1785].log_data[0].total := 300.0, [1785].log_data[0].time := 300.0, [1785].log_data[0].minminute := 5, [1785].log_data[0].maxminute := 5, [1785].log_data[0].valid := 1, [1785].log_data[1].valid := 1, [1785].log_data[2].valid := 1, [1785].log_data[3].valid := 1, [1785].log_data[4].valid := 1, [1785].log_data[5].valid := 1,
        [1785].log_data[6].valid := 1, [1785].log_data[7].valid := 1, [1785].log_data[8].valid := 1, [1785].log_data[9].valid := 1, [1785].log_data[10].valid := 1, [1785].log_data[11].valid := 1, [1785].log_data[12].valid := 1, [1785].log_data[13].valid := 1, [1785].log_data[14].valid := 1, [1785].log_data[15].valid := 1, [1785].log_data[16].valid := 1, [1785].log_data[17].valid := 1, [1785].log_data[18].valid := 1, [1785].log_data[19].valid := 1, [1785].time.Year := 2023, [1785].time.Month := 1, [1785].time.Day := 15, [1785].time.Hour := 21, [1785].time.Minute := 9, [1785].time.Second := 59, [1786].log_data[0].min := 1.0, [1786].log_data[0].max := 1.0, [1786].log_data[0].total := 300.0, [1786].log_data[0].time := 300.0, [1786].log_data[0].minminute := 10, [1786].log_data[0].maxminute := 10, [1786].log_data[0].valid := 1, [1786].log_data[1].valid := 1, [1786].log_data[2].valid := 1, [1786].log_data[3].valid := 1, [1786].log_data[4].valid := 1, [1786].log_data[5].valid := 1, [1786].log_data[6].valid := 1, [1786].log_data[7].valid := 1, [1786].log_data[8].valid := 1, [1786].log_data[9].valid := 1, [1786].log_data[10].valid := 1, [1786].log_data[11].valid := 1, [1786].log_data[12].valid := 1, [1786].log_data[13].valid := 1, [1786].log_data[14].valid := 1, [1786].log_data[15].valid := 1, [1786].log_data[16].valid := 1, [1786].log_data[17].valid := 1, [1786].log_data[18].valid := 1, [1786].log_data[19].valid := 1, [1786].time.Year := 2023, [1786].time.Month := 1, [1786].time.Day := 15, [1786].time.Hour := 21, [1786].time.Minute := 14, [1786].time.Second := 59, [1787].log_data[0].min := 1.0, [1787].log_data[0].max := 1.0, [1787].log_data[0].total := 300.0, [1787].log_data[0].time := 300.0, [1787].log_data[0].minminute := 15, [1787].log_data[0].maxminute := 15, [1787].log_data[0].valid := 1, [1787].log_data[1].valid := 1,
        [1787].log_data[2].valid := 1, [1787].log_data[3].valid := 1, [1787].log_data[4].valid := 1, [1787].log_data[5].valid := 1, [1787].log_data[6].valid := 1, [1787].log_data[7].valid := 1, [1787].log_data[8].valid := 1, [1787].log_data[9].valid := 1, [1787].log_data[10].valid := 1, [1787].log_data[11].valid := 1, [1787].log_data[12].valid := 1, [1787].log_data[13].valid := 1, [1787].log_data[14].valid := 1, [1787].log_data[15].valid := 1, [1787].log_data[16].valid := 1, [1787].log_data[17].valid := 1, [1787].log_data[18].valid := 1, [1787].log_data[19].valid := 1, [1787].time.Year := 2023, [1787].time.Month := 1, [1787].time.Day := 15, [1787].time.Hour := 21, [1787].time.Minute := 19, [1787].time.Second := 59, [1788].log_data[0].min := 1.0, [1788].log_data[0].max := 1.0, [1788].log_data[0].total := 300.0, [1788].log_data[0].time := 300.0, [1788].log_data[0].minminute := 20, [1788].log_data[0].maxminute := 20, [1788].log_data[0].valid := 1, [1788].log_data[1].valid := 1, [1788].log_data[2].valid := 1, [1788].log_data[3].valid := 1, [1788].log_data[4].valid := 1, [1788].log_data[5].valid := 1, [1788].log_data[6].valid := 1, [1788].log_data[7].valid := 1, [1788].log_data[8].valid := 1, [1788].log_data[9].valid := 1, [1788].log_data[10].valid := 1, [1788].log_data[11].valid := 1, [1788].log_data[12].valid := 1, [1788].log_data[13].valid := 1, [1788].log_data[14].valid := 1, [1788].log_data[15].valid := 1, [1788].log_data[16].valid := 1, [1788].log_data[17].valid := 1, [1788].log_data[18].valid := 1, [1788].log_data[19].valid := 1, [1788].time.Year := 2023, [1788].time.Month := 1, [1788].time.Day := 15, [1788].time.Hour := 21, [1788].time.Minute := 24, [1788].time.Second := 59, [1789].log_data[0].min := 1.0, [1789].log_data[0].max := 1.0, [1789].log_data[0].total := 300.0, [1789].log_data[0].time := 300.0,
        [1789].log_data[0].minminute := 25, [1789].log_data[0].maxminute := 25, [1789].log_data[0].valid := 1, [1789].log_data[1].valid := 1, [1789].log_data[2].valid := 1, [1789].log_data[3].valid := 1, [1789].log_data[4].valid := 1, [1789].log_data[5].valid := 1, [1789].log_data[6].valid := 1, [1789].log_data[7].valid := 1, [1789].log_data[8].valid := 1, [1789].log_data[9].valid := 1, [1789].log_data[10].valid := 1, [1789].log_data[11].valid := 1, [1789].log_data[12].valid := 1, [1789].log_data[13].valid := 1, [1789].log_data[14].valid := 1, [1789].log_data[15].valid := 1, [1789].log_data[16].valid := 1, [1789].log_data[17].valid := 1, [1789].log_data[18].valid := 1, [1789].log_data[19].valid := 1, [1789].time.Year := 2023, [1789].time.Month := 1, [1789].time.Day := 15, [1789].time.Hour := 21, [1789].time.Minute := 29, [1789].time.Second := 59, [1790].log_data[0].min := 1.0, [1790].log_data[0].max := 1.0, [1790].log_data[0].total := 300.0, [1790].log_data[0].time := 300.0, [1790].log_data[0].minminute := 30, [1790].log_data[0].maxminute := 30, [1790].log_data[0].valid := 1, [1790].log_data[1].valid := 1, [1790].log_data[2].valid := 1, [1790].log_data[3].valid := 1, [1790].log_data[4].valid := 1, [1790].log_data[5].valid := 1, [1790].log_data[6].valid := 1, [1790].log_data[7].valid := 1, [1790].log_data[8].valid := 1, [1790].log_data[9].valid := 1, [1790].log_data[10].valid := 1, [1790].log_data[11].valid := 1, [1790].log_data[12].valid := 1, [1790].log_data[13].valid := 1, [1790].log_data[14].valid := 1, [1790].log_data[15].valid := 1, [1790].log_data[16].valid := 1, [1790].log_data[17].valid := 1, [1790].log_data[18].valid := 1, [1790].log_data[19].valid := 1, [1790].time.Year := 2023, [1790].time.Month := 1, [1790].time.Day := 15, [1790].time.Hour := 21, [1790].time.Minute := 34, [1790].time.Second := 59,
        [1791].log_data[0].min := 1.0, [1791].log_data[0].max := 1.0, [1791].log_data[0].total := 300.0, [1791].log_data[0].time := 300.0, [1791].log_data[0].minminute := 35, [1791].log_data[0].maxminute := 35, [1791].log_data[0].valid := 1, [1791].log_data[1].valid := 1, [1791].log_data[2].valid := 1, [1791].log_data[3].valid := 1, [1791].log_data[4].valid := 1, [1791].log_data[5].valid := 1, [1791].log_data[6].valid := 1, [1791].log_data[7].valid := 1, [1791].log_data[8].valid := 1, [1791].log_data[9].valid := 1, [1791].log_data[10].valid := 1, [1791].log_data[11].valid := 1, [1791].log_data[12].valid := 1, [1791].log_data[13].valid := 1, [1791].log_data[14].valid := 1, [1791].log_data[15].valid := 1, [1791].log_data[16].valid := 1, [1791].log_data[17].valid := 1, [1791].log_data[18].valid := 1, [1791].log_data[19].valid := 1, [1791].time.Year := 2023, [1791].time.Month := 1, [1791].time.Day := 15, [1791].time.Hour := 21, [1791].time.Minute := 39, [1791].time.Second := 59, [1792].log_data[0].min := 1.0, [1792].log_data[0].max := 1.0, [1792].log_data[0].total := 300.0, [1792].log_data[0].time := 300.0, [1792].log_data[0].minminute := 40, [1792].log_data[0].maxminute := 40, [1792].log_data[0].valid := 1, [1792].log_data[1].valid := 1, [1792].log_data[2].valid := 1, [1792].log_data[3].valid := 1, [1792].log_data[4].valid := 1, [1792].log_data[5].valid := 1, [1792].log_data[6].valid := 1, [1792].log_data[7].valid := 1, [1792].log_data[8].valid := 1, [1792].log_data[9].valid := 1, [1792].log_data[10].valid := 1, [1792].log_data[11].valid := 1, [1792].log_data[12].valid := 1, [1792].log_data[13].valid := 1, [1792].log_data[14].valid := 1, [1792].log_data[15].valid := 1, [1792].log_data[16].valid := 1, [1792].log_data[17].valid := 1, [1792].log_data[18].valid := 1, [1792].log_data[19].valid := 1, [1792].time.Year := 2023, [1792].time.Month := 1,
        [1792].time.Day := 15, [1792].time.Hour := 21, [1792].time.Minute := 44, [1792].time.Second := 59, [1793].log_data[0].min := 1.0, [1793].log_data[0].max := 1.0, [1793].log_data[0].total := 300.0, [1793].log_data[0].time := 300.0, [1793].log_data[0].minminute := 45, [1793].log_data[0].maxminute := 45, [1793].log_data[0].valid := 1, [1793].log_data[1].valid := 1, [1793].log_data[2].valid := 1, [1793].log_data[3].valid := 1, [1793].log_data[4].valid := 1, [1793].log_data[5].valid := 1, [1793].log_data[6].valid := 1, [1793].log_data[7].valid := 1, [1793].log_data[8].valid := 1, [1793].log_data[9].valid := 1, [1793].log_data[10].valid := 1, [1793].log_data[11].valid := 1, [1793].log_data[12].valid := 1, [1793].log_data[13].valid := 1, [1793].log_data[14].valid := 1, [1793].log_data[15].valid := 1, [1793].log_data[16].valid := 1, [1793].log_data[17].valid := 1, [1793].log_data[18].valid := 1, [1793].log_data[19].valid := 1, [1793].time.Year := 2023, [1793].time.Month := 1, [1793].time.Day := 15, [1793].time.Hour := 21, [1793].time.Minute := 49, [1793].time.Second := 59, [1794].log_data[0].min := 1.0, [1794].log_data[0].max := 1.0, [1794].log_data[0].total := 300.0, [1794].log_data[0].time := 300.0, [1794].log_data[0].minminute := 50, [1794].log_data[0].maxminute := 50, [1794].log_data[0].valid := 1, [1794].log_data[1].valid := 1, [1794].log_data[2].valid := 1, [1794].log_data[3].valid := 1, [1794].log_data[4].valid := 1, [1794].log_data[5].valid := 1, [1794].log_data[6].valid := 1, [1794].log_data[7].valid := 1, [1794].log_data[8].valid := 1, [1794].log_data[9].valid := 1, [1794].log_data[10].valid := 1, [1794].log_data[11].valid := 1, [1794].log_data[12].valid := 1, [1794].log_data[13].valid := 1, [1794].log_data[14].valid := 1, [1794].log_data[15].valid := 1, [1794].log_data[16].valid := 1, [1794].log_data[17].valid := 1,
        [1794].log_data[18].valid := 1, [1794].log_data[19].valid := 1, [1794].time.Year := 2023, [1794].time.Month := 1, [1794].time.Day := 15, [1794].time.Hour := 21, [1794].time.Minute := 54, [1794].time.Second := 59, [1795].log_data[0].min := 1.0, [1795].log_data[0].max := 1.0, [1795].log_data[0].total := 300.0, [1795].log_data[0].time := 300.0, [1795].log_data[0].minminute := 55, [1795].log_data[0].maxminute := 55, [1795].log_data[0].valid := 1, [1795].log_data[1].valid := 1, [1795].log_data[2].valid := 1, [1795].log_data[3].valid := 1, [1795].log_data[4].valid := 1, [1795].log_data[5].valid := 1, [1795].log_data[6].valid := 1, [1795].log_data[7].valid := 1, [1795].log_data[8].valid := 1, [1795].log_data[9].valid := 1, [1795].log_data[10].valid := 1, [1795].log_data[11].valid := 1, [1795].log_data[12].valid := 1, [1795].log_data[13].valid := 1, [1795].log_data[14].valid := 1, [1795].log_data[15].valid := 1, [1795].log_data[16].valid := 1, [1795].log_data[17].valid := 1, [1795].log_data[18].valid := 1, [1795].log_data[19].valid := 1, [1795].time.Year := 2023, [1795].time.Month := 1, [1795].time.Day := 15, [1795].time.Hour := 21, [1795].time.Minute := 59, [1795].time.Second := 59, [1796].log_data[0].min := 1.0, [1796].log_data[0].max := 1.0, [1796].log_data[0].total := 299.5, [1796].log_data[0].time := 299.5, [1796].log_data[0].valid := 1, [1796].log_data[1].valid := 1, [1796].log_data[2].valid := 1, [1796].log_data[3].valid := 1, [1796].log_data[4].valid := 1, [1796].log_data[5].valid := 1, [1796].log_data[6].valid := 1, [1796].log_data[7].valid := 1, [1796].log_data[8].valid := 1, [1796].log_data[9].valid := 1, [1796].log_data[10].valid := 1, [1796].log_data[11].valid := 1, [1796].log_data[12].valid := 1, [1796].log_data[13].valid := 1, [1796].log_data[14].valid := 1, [1796].log_data[15].valid := 1,
        [1796].log_data[16].valid := 1, [1796].log_data[17].valid := 1, [1796].log_data[18].valid := 1, [1796].log_data[19].valid := 1, [1796].time.Year := 2023, [1796].time.Month := 1, [1796].time.Day := 15, [1796].time.Hour := 22, [1796].time.Minute := 4, [1796].time.Second := 59, [1797].log_data[0].min := 1.0, [1797].log_data[0].max := 1.0, [1797].log_data[0].total := 300.0, [1797].log_data[0].time := 300.0, [1797].log_data[0].minminute := 5, [1797].log_data[0].maxminute := 5, [1797].log_data[0].valid := 1, [1797].log_data[1].valid := 1, [1797].log_data[2].valid := 1, [1797].log_data[3].valid := 1, [1797].log_data[4].valid := 1, [1797].log_data[5].valid := 1, [1797].log_data[6].valid := 1, [1797].log_data[7].valid := 1, [1797].log_data[8].valid := 1, [1797].log_data[9].valid := 1, [1797].log_data[10].valid := 1, [1797].log_data[11].valid := 1, [1797].log_data[12].valid := 1, [1797].log_data[13].valid := 1, [1797].log_data[14].valid := 1, [1797].log_data[15].valid := 1, [1797].log_data[16].valid := 1, [1797].log_data[17].valid := 1, [1797].log_data[18].valid := 1, [1797].log_data[19].valid := 1, [1797].time.Year := 2023, [1797].time.Month := 1, [1797].time.Day := 15, [1797].time.Hour := 22, [1797].time.Minute := 9, [1797].time.Second := 59, [1798].log_data[0].min := 1.0, [1798].log_data[0].max := 1.0, [1798].log_data[0].total := 300.0, [1798].log_data[0].time := 300.0, [1798].log_data[0].minminute := 10, [1798].log_data[0].maxminute := 10, [1798].log_data[0].valid := 1, [1798].log_data[1].valid := 1, [1798].log_data[2].valid := 1, [1798].log_data[3].valid := 1, [1798].log_data[4].valid := 1, [1798].log_data[5].valid := 1, [1798].log_data[6].valid := 1, [1798].log_data[7].valid := 1, [1798].log_data[8].valid := 1, [1798].log_data[9].valid := 1, [1798].log_data[10].valid := 1, [1798].log_data[11].valid := 1,
        [1798].log_data[12].valid := 1, [1798].log_data[13].valid := 1, [1798].log_data[14].valid := 1, [1798].log_data[15].valid := 1, [1798].log_data[16].valid := 1, [1798].log_data[17].valid := 1, [1798].log_data[18].valid := 1, [1798].log_data[19].valid := 1, [1798].time.Year := 2023, [1798].time.Month := 1, [1798].time.Day := 15, [1798].time.Hour := 22, [1798].time.Minute := 14, [1798].time.Second := 59, [1799].log_data[0].min := 1.0, [1799].log_data[0].max := 1.0, [1799].log_data[0].total := 300.0, [1799].log_data[0].time := 300.0, [1799].log_data[0].minminute := 15, [1799].log_data[0].maxminute := 15, [1799].log_data[0].valid := 1, [1799].log_data[1].valid := 1, [1799].log_data[2].valid := 1, [1799].log_data[3].valid := 1, [1799].log_data[4].valid := 1, [1799].log_data[5].valid := 1, [1799].log_data[6].valid := 1, [1799].log_data[7].valid := 1, [1799].log_data[8].valid := 1, [1799].log_data[9].valid := 1, [1799].log_data[10].valid := 1, [1799].log_data[11].valid := 1, [1799].log_data[12].valid := 1, [1799].log_data[13].valid := 1, [1799].log_data[14].valid := 1, [1799].log_data[15].valid := 1, [1799].log_data[16].valid := 1, [1799].log_data[17].valid := 1, [1799].log_data[18].valid := 1, [1799].log_data[19].valid := 1, [1799].time.Year := 2023, [1799].time.Month := 1, [1799].time.Day := 15, [1799].time.Hour := 22, [1799].time.Minute := 19, [1799].time.Second := 59, [1800].log_data[0].min := 1.0, [1800].log_data[0].max := 1.0, [1800].log_data[0].total := 300.0, [1800].log_data[0].time := 300.0, [1800].log_data[0].minminute := 20, [1800].log_data[0].maxminute := 20, [1800].log_data[0].valid := 1, [1800].log_data[1].valid := 1, [1800].log_data[2].valid := 1, [1800].log_data[3].valid := 1, [1800].log_data[4].valid := 1, [1800].log_data[5].valid := 1, [1800].log_data[6].valid := 1, [1800].log_data[7].valid := 1,
        [1800].log_data[8].valid := 1, [1800].log_data[9].valid := 1, [1800].log_data[10].valid := 1, [1800].log_data[11].valid := 1, [1800].log_data[12].valid := 1, [1800].log_data[13].valid := 1, [1800].log_data[14].valid := 1, [1800].log_data[15].valid := 1, [1800].log_data[16].valid := 1, [1800].log_data[17].valid := 1, [1800].log_data[18].valid := 1, [1800].log_data[19].valid := 1, [1800].time.Year := 2023, [1800].time.Month := 1, [1800].time.Day := 15, [1800].time.Hour := 22, [1800].time.Minute := 24, [1800].time.Second := 59, [1801].log_data[0].min := 1.0, [1801].log_data[0].max := 1.0, [1801].log_data[0].total := 300.0, [1801].log_data[0].time := 300.0, [1801].log_data[0].minminute := 25, [1801].log_data[0].maxminute := 25, [1801].log_data[0].valid := 1, [1801].log_data[1].valid := 1, [1801].log_data[2].valid := 1, [1801].log_data[3].valid := 1, [1801].log_data[4].valid := 1, [1801].log_data[5].valid := 1, [1801].log_data[6].valid := 1, [1801].log_data[7].valid := 1, [1801].log_data[8].valid := 1, [1801].log_data[9].valid := 1, [1801].log_data[10].valid := 1, [1801].log_data[11].valid := 1, [1801].log_data[12].valid := 1, [1801].log_data[13].valid := 1, [1801].log_data[14].valid := 1, [1801].log_data[15].valid := 1, [1801].log_data[16].valid := 1, [1801].log_data[17].valid := 1, [1801].log_data[18].valid := 1, [1801].log_data[19].valid := 1, [1801].time.Year := 2023, [1801].time.Month := 1, [1801].time.Day := 15, [1801].time.Hour := 22, [1801].time.Minute := 29, [1801].time.Second := 59, [1802].log_data[0].min := 1.0, [1802].log_data[0].max := 1.0, [1802].log_data[0].total := 300.0, [1802].log_data[0].time := 300.0, [1802].log_data[0].minminute := 30, [1802].log_data[0].maxminute := 30, [1802].log_data[0].valid := 1, [1802].log_data[1].valid := 1, [1802].log_data[2].valid := 1, [1802].log_data[3].valid := 1,
        [1802].log_data[4].valid := 1, [1802].log_data[5].valid := 1, [1802].log_data[6].valid := 1, [1802].log_data[7].valid := 1, [1802].log_data[8].valid := 1, [1802].log_data[9].valid := 1, [1802].log_data[10].valid := 1, [1802].log_data[11].valid := 1, [1802].log_data[12].valid := 1, [1802].log_data[13].valid := 1, [1802].log_data[14].valid := 1, [1802].log_data[15].valid := 1, [1802].log_data[16].valid := 1, [1802].log_data[17].valid := 1, [1802].log_data[18].valid := 1, [1802].log_data[19].valid := 1, [1802].time.Year := 2023, [1802].time.Month := 1, [1802].time.Day := 15, [1802].time.Hour := 22, [1802].time.Minute := 34, [1802].time.Second := 59, [1803].log_data[0].min := 1.0, [1803].log_data[0].max := 1.0, [1803].log_data[0].total := 300.0, [1803].log_data[0].time := 300.0, [1803].log_data[0].minminute := 35, [1803].log_data[0].maxminute := 35, [1803].log_data[0].valid := 1, [1803].log_data[1].valid := 1, [1803].log_data[2].valid := 1, [1803].log_data[3].valid := 1, [1803].log_data[4].valid := 1, [1803].log_data[5].valid := 1, [1803].log_data[6].valid := 1, [1803].log_data[7].valid := 1, [1803].log_data[8].valid := 1, [1803].log_data[9].valid := 1, [1803].log_data[10].valid := 1, [1803].log_data[11].valid := 1, [1803].log_data[12].valid := 1, [1803].log_data[13].valid := 1, [1803].log_data[14].valid := 1, [1803].log_data[15].valid := 1, [1803].log_data[16].valid := 1, [1803].log_data[17].valid := 1, [1803].log_data[18].valid := 1, [1803].log_data[19].valid := 1, [1803].time.Year := 2023, [1803].time.Month := 1, [1803].time.Day := 15, [1803].time.Hour := 22, [1803].time.Minute := 39, [1803].time.Second := 59, [1804].log_data[0].min := 1.0, [1804].log_data[0].max := 1.0, [1804].log_data[0].total := 300.0, [1804].log_data[0].time := 300.0, [1804].log_data[0].minminute := 40, [1804].log_data[0].maxminute := 40,
        [1804].log_data[0].valid := 1, [1804].log_data[1].valid := 1, [1804].log_data[2].valid := 1, [1804].log_data[3].valid := 1, [1804].log_data[4].valid := 1, [1804].log_data[5].valid := 1, [1804].log_data[6].valid := 1, [1804].log_data[7].valid := 1, [1804].log_data[8].valid := 1, [1804].log_data[9].valid := 1, [1804].log_data[10].valid := 1, [1804].log_data[11].valid := 1, [1804].log_data[12].valid := 1, [1804].log_data[13].valid := 1, [1804].log_data[14].valid := 1, [1804].log_data[15].valid := 1, [1804].log_data[16].valid := 1, [1804].log_data[17].valid := 1, [1804].log_data[18].valid := 1, [1804].log_data[19].valid := 1, [1804].time.Year := 2023, [1804].time.Month := 1, [1804].time.Day := 15, [1804].time.Hour := 22, [1804].time.Minute := 44, [1804].time.Second := 59, [1805].log_data[0].min := 1.0, [1805].log_data[0].max := 1.0, [1805].log_data[0].total := 300.0, [1805].log_data[0].time := 300.0, [1805].log_data[0].minminute := 45, [1805].log_data[0].maxminute := 45, [1805].log_data[0].valid := 1, [1805].log_data[1].valid := 1, [1805].log_data[2].valid := 1, [1805].log_data[3].valid := 1, [1805].log_data[4].valid := 1, [1805].log_data[5].valid := 1, [1805].log_data[6].valid := 1, [1805].log_data[7].valid := 1, [1805].log_data[8].valid := 1, [1805].log_data[9].valid := 1, [1805].log_data[10].valid := 1, [1805].log_data[11].valid := 1, [1805].log_data[12].valid := 1, [1805].log_data[13].valid := 1, [1805].log_data[14].valid := 1, [1805].log_data[15].valid := 1, [1805].log_data[16].valid := 1, [1805].log_data[17].valid := 1, [1805].log_data[18].valid := 1, [1805].log_data[19].valid := 1, [1805].time.Year := 2023, [1805].time.Month := 1, [1805].time.Day := 15, [1805].time.Hour := 22, [1805].time.Minute := 49, [1805].time.Second := 59, [1806].log_data[0].min := 1.0, [1806].log_data[0].max := 1.0,
        [1806].log_data[0].total := 300.0, [1806].log_data[0].time := 300.0, [1806].log_data[0].minminute := 50, [1806].log_data[0].maxminute := 50, [1806].log_data[0].valid := 1, [1806].log_data[1].valid := 1, [1806].log_data[2].valid := 1, [1806].log_data[3].valid := 1, [1806].log_data[4].valid := 1, [1806].log_data[5].valid := 1, [1806].log_data[6].valid := 1, [1806].log_data[7].valid := 1, [1806].log_data[8].valid := 1, [1806].log_data[9].valid := 1, [1806].log_data[10].valid := 1, [1806].log_data[11].valid := 1, [1806].log_data[12].valid := 1, [1806].log_data[13].valid := 1, [1806].log_data[14].valid := 1, [1806].log_data[15].valid := 1, [1806].log_data[16].valid := 1, [1806].log_data[17].valid := 1, [1806].log_data[18].valid := 1, [1806].log_data[19].valid := 1, [1806].time.Year := 2023, [1806].time.Month := 1, [1806].time.Day := 15, [1806].time.Hour := 22, [1806].time.Minute := 54, [1806].time.Second := 59, [1807].log_data[0].min := 1.0, [1807].log_data[0].max := 1.0, [1807].log_data[0].total := 300.0, [1807].log_data[0].time := 300.0, [1807].log_data[0].minminute := 55, [1807].log_data[0].maxminute := 55, [1807].log_data[0].valid := 1, [1807].log_data[1].valid := 1, [1807].log_data[2].valid := 1, [1807].log_data[3].valid := 1, [1807].log_data[4].valid := 1, [1807].log_data[5].valid := 1, [1807].log_data[6].valid := 1, [1807].log_data[7].valid := 1, [1807].log_data[8].valid := 1, [1807].log_data[9].valid := 1, [1807].log_data[10].valid := 1, [1807].log_data[11].valid := 1, [1807].log_data[12].valid := 1, [1807].log_data[13].valid := 1, [1807].log_data[14].valid := 1, [1807].log_data[15].valid := 1, [1807].log_data[16].valid := 1, [1807].log_data[17].valid := 1, [1807].log_data[18].valid := 1, [1807].log_data[19].valid := 1, [1807].time.Year := 2023, [1807].time.Month := 1, [1807].time.Day := 15, [1807].time.Hour := 22,
        [1807].time.Minute := 59, [1807].time.Second := 59, [1808].log_data[0].min := 1.0, [1808].log_data[0].max := 1.0, [1808].log_data[0].total := 300.0, [1808].log_data[0].time := 300.0, [1808].log_data[0].valid := 1, [1808].log_data[1].valid := 1, [1808].log_data[2].valid := 1, [1808].log_data[3].valid := 1, [1808].log_data[4].valid := 1, [1808].log_data[5].valid := 1, [1808].log_data[6].valid := 1, [1808].log_data[7].valid := 1, [1808].log_data[8].valid := 1, [1808].log_data[9].valid := 1, [1808].log_data[10].valid := 1, [1808].log_data[11].valid := 1, [1808].log_data[12].valid := 1, [1808].log_data[13].valid := 1, [1808].log_data[14].valid := 1, [1808].log_data[15].valid := 1, [1808].log_data[16].valid := 1, [1808].log_data[17].valid := 1, [1808].log_data[18].valid := 1, [1808].log_data[19].valid := 1, [1808].time.Year := 2023, [1808].time.Month := 1, [1808].time.Day := 15, [1808].time.Hour := 23, [1808].time.Minute := 4, [1808].time.Second := 59, [1809].log_data[0].min := 1.0, [1809].log_data[0].max := 1.0, [1809].log_data[0].total := 300.0, [1809].log_data[0].time := 300.0, [1809].log_data[0].minminute := 5, [1809].log_data[0].maxminute := 5, [1809].log_data[0].valid := 1, [1809].log_data[1].valid := 1, [1809].log_data[2].valid := 1, [1809].log_data[3].valid := 1, [1809].log_data[4].valid := 1, [1809].log_data[5].valid := 1, [1809].log_data[6].valid := 1, [1809].log_data[7].valid := 1, [1809].log_data[8].valid := 1, [1809].log_data[9].valid := 1, [1809].log_data[10].valid := 1, [1809].log_data[11].valid := 1, [1809].log_data[12].valid := 1, [1809].log_data[13].valid := 1, [1809].log_data[14].valid := 1, [1809].log_data[15].valid := 1, [1809].log_data[16].valid := 1, [1809].log_data[17].valid := 1, [1809].log_data[18].valid := 1, [1809].log_data[19].valid := 1, [1809].time.Year := 2023, [1809].time.Month := 1,
